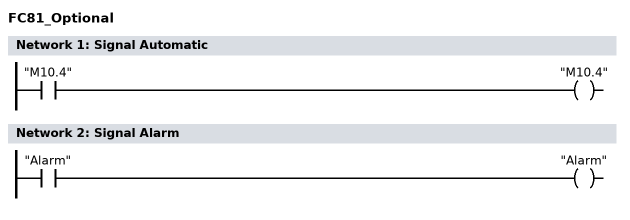
   RUNG wire#powerrail
      Contact( "M10.4" )
      Coil( "M10.4" )
   END_RUNG
   // the same network as SCL:
   "M10.4" := "M10.4";
END_REGION

REGION Network 2: Signal Alarm
   RUNG wire#powerrail
      Contact( "Alarm" )
      Coil( "Alarm" )
   END_RUNG
   // the same network as SCL:
   "Alarm" := "Alarm";
END_REGION
END_FUNCTION

FUNCTION "FC82_Conveyor_2_IN_2_OUT" : Void   // FC82, LAD
TITLE = Conveyor_2_IN_2_OUT
{ S7_Optimized_Access := 'TRUE' }
VERSION : 0.1
// stored: AutoNumber false, IsIECCheckEnabled false, SetENOAutomatically false, UDAEnableTagReadback false
   VAR_TEMP   // added for the SCL form of the ladder/FBD networks
      _w1 : Bool;
      _w2 : Bool;
   END_VAR
BEGIN

REGION Network 1: Manual operation for conveyor
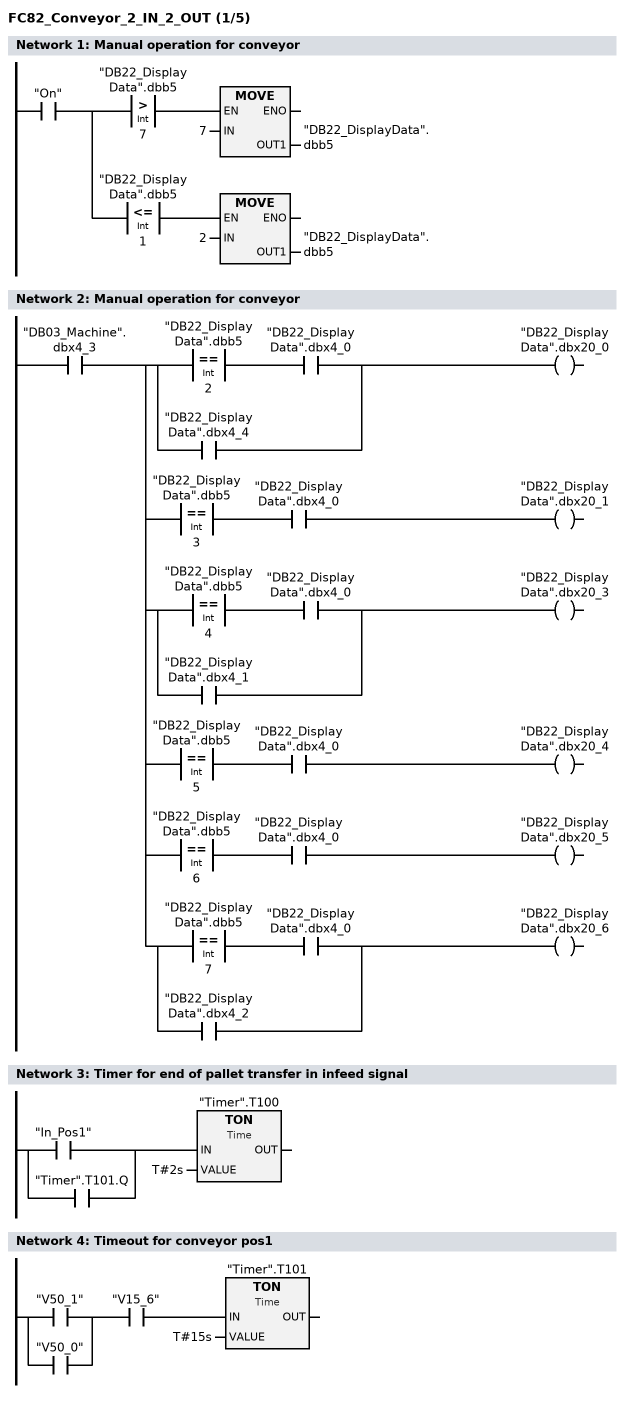
   RUNG wire#powerrail
      Contact( "On" )
      wire#w1
      { S7_Templates := "SrcType := Int" } GT_Contact(in1 := "DB22_DisplayData".dbb5, in2 := 7)
      { S7_GenerateENO := "TRUE" } Move(in := 7, out1 => "DB22_DisplayData".dbb5)
   END_RUNG
   RUNG wire#w1
      { S7_Templates := "SrcType := Int" } LE_Contact(in1 := "DB22_DisplayData".dbb5, in2 := 1)
      { S7_GenerateENO := "TRUE" } Move(in := 2, out1 => "DB22_DisplayData".dbb5)
   END_RUNG
   // the same network as SCL:
   IF "On" AND ("DB22_DisplayData".dbb5 > 7) THEN "DB22_DisplayData".dbb5 := 7; END_IF;
   IF "On" AND ("DB22_DisplayData".dbb5 <= 1) THEN "DB22_DisplayData".dbb5 := 2; END_IF;
END_REGION

REGION Network 2: Manual operation for conveyor
   RUNG wire#powerrail
      Contact( "DB03_Machine".dbx4_3 )
      wire#w1
      { S7_Templates := "SrcType := Int" } EQ_Contact(in1 := "DB22_DisplayData".dbb5, in2 := 2)
      Contact( "DB22_DisplayData".dbx4_0 )
      wire#w2
      Coil( "DB22_DisplayData".dbx20_0 )
   END_RUNG
   RUNG wire#w1
      Contact( "DB22_DisplayData".dbx4_4 )
   END_RUNG wire#w2
   RUNG wire#w1
      { S7_Templates := "SrcType := Int" } EQ_Contact(in1 := "DB22_DisplayData".dbb5, in2 := 3)
      Contact( "DB22_DisplayData".dbx4_0 )
      Coil( "DB22_DisplayData".dbx20_1 )
   END_RUNG
   RUNG wire#w1
      { S7_Templates := "SrcType := Int" } EQ_Contact(in1 := "DB22_DisplayData".dbb5, in2 := 4)
      Contact( "DB22_DisplayData".dbx4_0 )
      wire#w3
      Coil( "DB22_DisplayData".dbx20_3 )
   END_RUNG
   RUNG wire#w1
      Contact( "DB22_DisplayData".dbx4_1 )
   END_RUNG wire#w3
   RUNG wire#w1
      { S7_Templates := "SrcType := Int" } EQ_Contact(in1 := "DB22_DisplayData".dbb5, in2 := 5)
      Contact( "DB22_DisplayData".dbx4_0 )
      Coil( "DB22_DisplayData".dbx20_4 )
   END_RUNG
   RUNG wire#w1
      { S7_Templates := "SrcType := Int" } EQ_Contact(in1 := "DB22_DisplayData".dbb5, in2 := 6)
      Contact( "DB22_DisplayData".dbx4_0 )
      Coil( "DB22_DisplayData".dbx20_5 )
   END_RUNG
   RUNG wire#w1
      { S7_Templates := "SrcType := Int" } EQ_Contact(in1 := "DB22_DisplayData".dbb5, in2 := 7)
      Contact( "DB22_DisplayData".dbx4_0 )
      wire#w4
      Coil( "DB22_DisplayData".dbx20_6 )
   END_RUNG
   RUNG wire#w1
      Contact( "DB22_DisplayData".dbx4_2 )
   END_RUNG wire#w4
   // the same network as SCL:
   "DB22_DisplayData".dbx20_0 := "DB03_Machine".dbx4_3 AND ((("DB22_DisplayData".dbb5 = 2) AND "DB22_DisplayData".dbx4_0) OR "DB22_DisplayData".dbx4_4);
   "DB22_DisplayData".dbx20_1 := "DB03_Machine".dbx4_3 AND ("DB22_DisplayData".dbb5 = 3) AND "DB22_DisplayData".dbx4_0;
   "DB22_DisplayData".dbx20_3 := "DB03_Machine".dbx4_3 AND ((("DB22_DisplayData".dbb5 = 4) AND "DB22_DisplayData".dbx4_0) OR "DB22_DisplayData".dbx4_1);
   "DB22_DisplayData".dbx20_4 := "DB03_Machine".dbx4_3 AND ("DB22_DisplayData".dbb5 = 5) AND "DB22_DisplayData".dbx4_0;
   "DB22_DisplayData".dbx20_5 := "DB03_Machine".dbx4_3 AND ("DB22_DisplayData".dbb5 = 6) AND "DB22_DisplayData".dbx4_0;
   "DB22_DisplayData".dbx20_6 := "DB03_Machine".dbx4_3 AND ((("DB22_DisplayData".dbb5 = 7) AND "DB22_DisplayData".dbx4_0) OR "DB22_DisplayData".dbx4_2);
END_REGION

REGION Network 3: Timer for end of pallet transfer in infeed signal
   "Timer".T100.TON(IN := "In_Pos1" OR "Timer".T101.Q, PT := T#2s);   // TON coil
END_REGION

REGION Network 4: Timeout for conveyor pos1
   "Timer".T101.TON(IN := ("V50_1" OR "V50_0") AND "V15_6", PT := T#15s);   // TON coil
END_REGION

REGION Network 5: Time to load with forklift
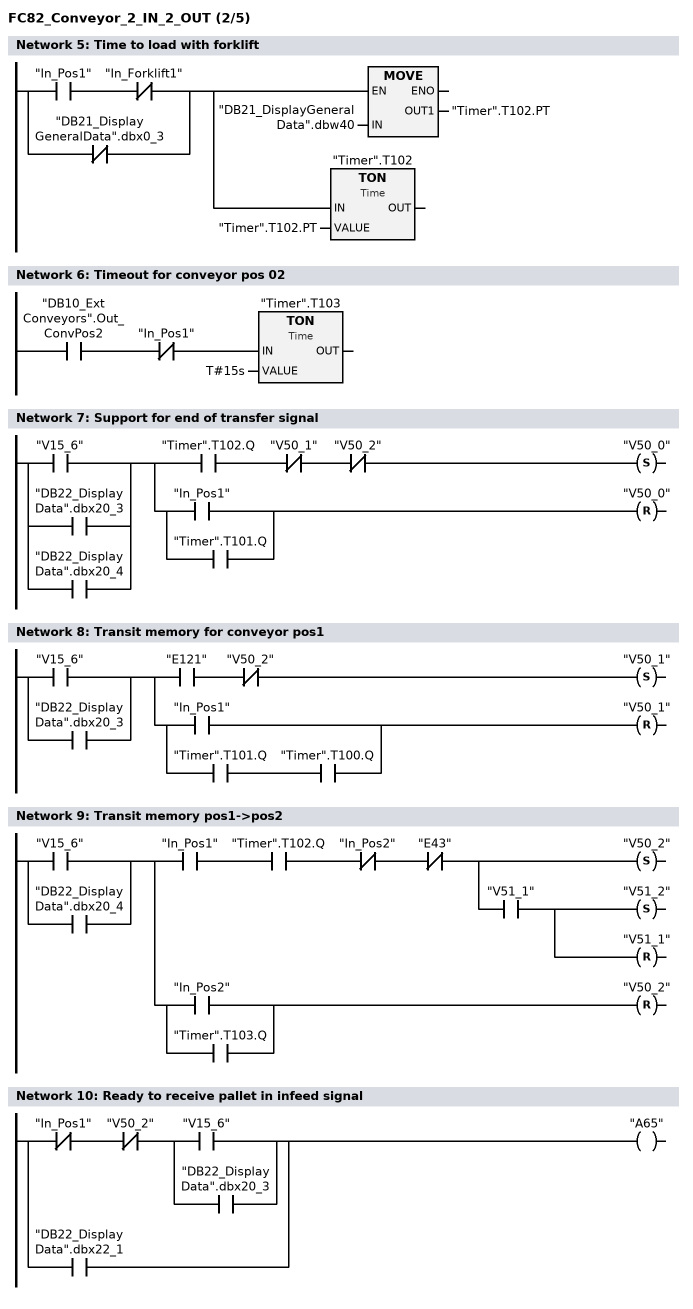
   #_w1 := ("In_Pos1" AND NOT "In_Forklift1") OR NOT "DB21_DisplayGeneralData".dbx0_3;
   IF #_w1 THEN "Timer".T102.PT := "DB21_DisplayGeneralData".dbw40; END_IF;
   "Timer".T102.TON(IN := #_w1, PT := "Timer".T102.PT);   // TON coil
END_REGION

REGION Network 6: Timeout for conveyor pos 02
   "Timer".T103.TON(IN := "DB10_ExtConveyors".Out_ConvPos2 AND NOT "In_Pos1", PT := T#15s);   // TON coil
END_REGION

REGION Network 7: Support for end of transfer signal
   RUNG wire#powerrail
      Contact( "V15_6" )
      wire#w1
      Contact( "Timer".T102.Q )
      I_Contact( "V50_1" )
      I_Contact( "V50_2" )
      S_Coil( "V50_0" )
   END_RUNG
   RUNG wire#powerrail
      Contact( "DB22_DisplayData".dbx20_3 )
   END_RUNG wire#w1
   RUNG wire#powerrail
      Contact( "DB22_DisplayData".dbx20_4 )
   END_RUNG wire#w1
   RUNG wire#w1
      Contact( "In_Pos1" )
      wire#w2
      R_Coil( "V50_0" )
   END_RUNG
   RUNG wire#w1
      Contact( "Timer".T101.Q )
   END_RUNG wire#w2
   // the same network as SCL:
   #_w1 := "V15_6" OR "DB22_DisplayData".dbx20_3 OR "DB22_DisplayData".dbx20_4;
   IF #_w1 AND "Timer".T102.Q AND NOT "V50_1" AND NOT "V50_2" THEN "V50_0" := TRUE; END_IF;
   IF #_w1 AND ("In_Pos1" OR "Timer".T101.Q) THEN "V50_0" := FALSE; END_IF;
END_REGION

REGION Network 8: Transit memory for conveyor pos1
   RUNG wire#powerrail
      Contact( "V15_6" )
      wire#w1
      Contact( "E121" )
      I_Contact( "V50_2" )
      S_Coil( "V50_1" )
   END_RUNG
   RUNG wire#powerrail
      Contact( "DB22_DisplayData".dbx20_3 )
   END_RUNG wire#w1
   RUNG wire#w1
      Contact( "In_Pos1" )
      wire#w2
      R_Coil( "V50_1" )
   END_RUNG
   RUNG wire#w1
      Contact( "Timer".T101.Q )
      Contact( "Timer".T100.Q )
   END_RUNG wire#w2
   // the same network as SCL:
   #_w1 := "V15_6" OR "DB22_DisplayData".dbx20_3;
   IF #_w1 AND "E121" AND NOT "V50_2" THEN "V50_1" := TRUE; END_IF;
   IF #_w1 AND ("In_Pos1" OR ("Timer".T101.Q AND "Timer".T100.Q)) THEN "V50_1" := FALSE; END_IF;
END_REGION

REGION Network 9: Transit memory pos1->pos2
   RUNG wire#powerrail
      Contact( "V15_6" )
      wire#w1
      Contact( "In_Pos1" )
      Contact( "Timer".T102.Q )
      I_Contact( "In_Pos2" )
      I_Contact( "E43" )
      wire#w2
      S_Coil( "V50_2" )
   END_RUNG
   RUNG wire#powerrail
      Contact( "DB22_DisplayData".dbx20_4 )
   END_RUNG wire#w1
   RUNG wire#w2
      Contact( "V51_1" )
      wire#w3
      S_Coil( "V51_2" )
   END_RUNG
   RUNG wire#w3
      R_Coil( "V51_1" )
   END_RUNG
   RUNG wire#w1
      Contact( "In_Pos2" )
      wire#w4
      R_Coil( "V50_2" )
   END_RUNG
   RUNG wire#w1
      Contact( "Timer".T103.Q )
   END_RUNG wire#w4
   // the same network as SCL:
   #_w1 := "V15_6" OR "DB22_DisplayData".dbx20_4;
   #_w2 := #_w1 AND "In_Pos1" AND "Timer".T102.Q AND NOT "In_Pos2" AND NOT "E43";
   IF #_w2 THEN "V50_2" := TRUE; END_IF;
   IF #_w2 AND "V51_1" THEN
       "V51_2" := TRUE;
       "V51_1" := FALSE;
   END_IF;
   IF #_w1 AND ("In_Pos2" OR "Timer".T103.Q) THEN "V50_2" := FALSE; END_IF;
END_REGION

REGION Network 10: Ready to receive pallet in infeed signal
   RUNG wire#powerrail
      I_Contact( "In_Pos1" )
      I_Contact( "V50_2" )
      wire#w1
      Contact( "V15_6" )
      wire#w2
      Coil( "A65" )
   END_RUNG
   RUNG wire#w1
      Contact( "DB22_DisplayData".dbx20_3 )
   END_RUNG wire#w2
   RUNG wire#powerrail
      Contact( "DB22_DisplayData".dbx22_1 )
   END_RUNG wire#w2
   // the same network as SCL:
   "A65" := (NOT "In_Pos1" AND NOT "V50_2" AND ("V15_6" OR "DB22_DisplayData".dbx20_3)) OR "DB22_DisplayData".dbx22_1;
END_REGION

REGION Network 11: End of pallet transfer in infeed signal
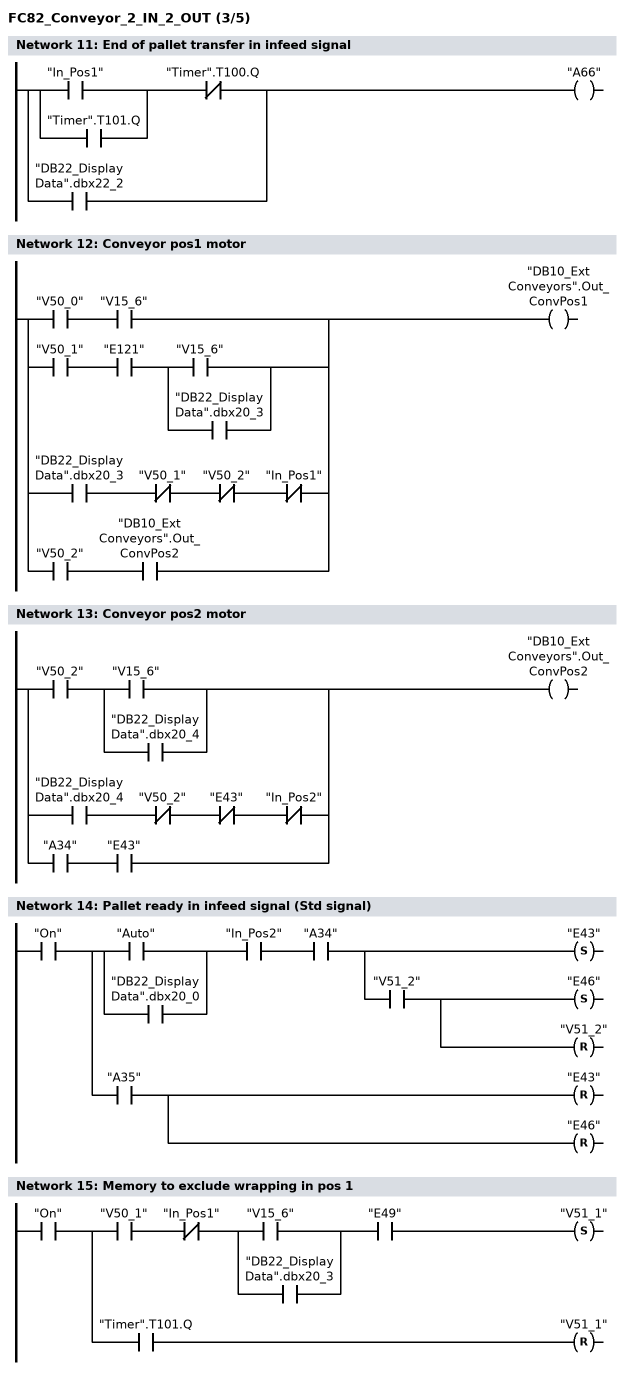
   RUNG wire#powerrail
      Contact( "In_Pos1" )
      wire#w1
      I_Contact( "Timer".T100.Q )
      wire#w2
      Coil( "A66" )
   END_RUNG
   RUNG wire#powerrail
      Contact( "Timer".T101.Q )
   END_RUNG wire#w1
   RUNG wire#powerrail
      Contact( "DB22_DisplayData".dbx22_2 )
   END_RUNG wire#w2
   // the same network as SCL:
   "A66" := (("In_Pos1" OR "Timer".T101.Q) AND NOT "Timer".T100.Q) OR "DB22_DisplayData".dbx22_2;
END_REGION

REGION Network 12: Conveyor pos1 motor
   RUNG wire#powerrail
      Contact( "V50_0" )
      Contact( "V15_6" )
      wire#w1
      Coil( "DB10_ExtConveyors".Out_ConvPos1 )
   END_RUNG
   RUNG wire#powerrail
      Contact( "V50_1" )
      Contact( "E121" )
      wire#w2
      Contact( "V15_6" )
   END_RUNG wire#w1
   RUNG wire#w2
      Contact( "DB22_DisplayData".dbx20_3 )
   END_RUNG wire#w1
   RUNG wire#powerrail
      Contact( "DB22_DisplayData".dbx20_3 )
      I_Contact( "V50_1" )
      I_Contact( "V50_2" )
      I_Contact( "In_Pos1" )
   END_RUNG wire#w1
   RUNG wire#powerrail
      Contact( "V50_2" )
      Contact( "DB10_ExtConveyors".Out_ConvPos2 )
   END_RUNG wire#w1
   // the same network as SCL:
   "DB10_ExtConveyors".Out_ConvPos1 := ("V50_0" AND "V15_6") OR ("V50_1" AND "E121" AND ("V15_6" OR "DB22_DisplayData".dbx20_3)) OR ("DB22_DisplayData".dbx20_3 AND NOT "V50_1" AND NOT "V50_2" AND NOT "In_Pos1") OR ("V50_2" AND "DB10_ExtConveyors".Out_ConvPos2);
END_REGION

REGION Network 13: Conveyor pos2 motor
   RUNG wire#powerrail
      Contact( "V50_2" )
      wire#w1
      Contact( "V15_6" )
      wire#w2
      Coil( "DB10_ExtConveyors".Out_ConvPos2 )
   END_RUNG
   RUNG wire#w1
      Contact( "DB22_DisplayData".dbx20_4 )
   END_RUNG wire#w2
   RUNG wire#powerrail
      Contact( "DB22_DisplayData".dbx20_4 )
      I_Contact( "V50_2" )
      I_Contact( "E43" )
      I_Contact( "In_Pos2" )
   END_RUNG wire#w2
   RUNG wire#powerrail
      Contact( "A34" )
      Contact( "E43" )
   END_RUNG wire#w2
   // the same network as SCL:
   "DB10_ExtConveyors".Out_ConvPos2 := ("V50_2" AND ("V15_6" OR "DB22_DisplayData".dbx20_4)) OR ("DB22_DisplayData".dbx20_4 AND NOT "V50_2" AND NOT "E43" AND NOT "In_Pos2") OR ("A34" AND "E43");
END_REGION

REGION Network 14: Pallet ready in infeed signal (Std signal)
   RUNG wire#powerrail
      Contact( "On" )
      wire#w1
      Contact( "Auto" )
      wire#w2
      Contact( "In_Pos2" )
      Contact( "A34" )
      wire#w3
      S_Coil( "E43" )
   END_RUNG
   RUNG wire#w1
      Contact( "DB22_DisplayData".dbx20_0 )
   END_RUNG wire#w2
   RUNG wire#w3
      Contact( "V51_2" )
      wire#w4
      S_Coil( "E46" )
   END_RUNG
   RUNG wire#w4
      R_Coil( "V51_2" )
   END_RUNG
   RUNG wire#w1
      Contact( "A35" )
      wire#w5
      R_Coil( "E43" )
   END_RUNG
   RUNG wire#w5
      R_Coil( "E46" )
   END_RUNG
   // the same network as SCL:
   #_w1 := "On" AND ("Auto" OR "DB22_DisplayData".dbx20_0) AND "In_Pos2" AND "A34";
   IF #_w1 THEN "E43" := TRUE; END_IF;
   IF #_w1 AND "V51_2" THEN
       "E46" := TRUE;
       "V51_2" := FALSE;
   END_IF;
   IF "On" AND "A35" THEN
       "E43" := FALSE;
       "E46" := FALSE;
   END_IF;
END_REGION

REGION Network 15: Memory to exclude wrapping in pos 1
   RUNG wire#powerrail
      Contact( "On" )
      wire#w1
      Contact( "V50_1" )
      I_Contact( "In_Pos1" )
      wire#w2
      Contact( "V15_6" )
      wire#w3
      Contact( "E49" )
      S_Coil( "V51_1" )
   END_RUNG
   RUNG wire#w2
      Contact( "DB22_DisplayData".dbx20_3 )
   END_RUNG wire#w3
   RUNG wire#w1
      Contact( "Timer".T101.Q )
      R_Coil( "V51_1" )
   END_RUNG
   // the same network as SCL:
   IF "On" AND "V50_1" AND NOT "In_Pos1" AND ("V15_6" OR "DB22_DisplayData".dbx20_3) AND "E49" THEN
       "V51_1" := TRUE;
   END_IF;
   IF "On" AND "Timer".T101.Q THEN "V51_1" := FALSE; END_IF;
END_REGION

REGION Network 16: Conveyor pos1 motor speed selection
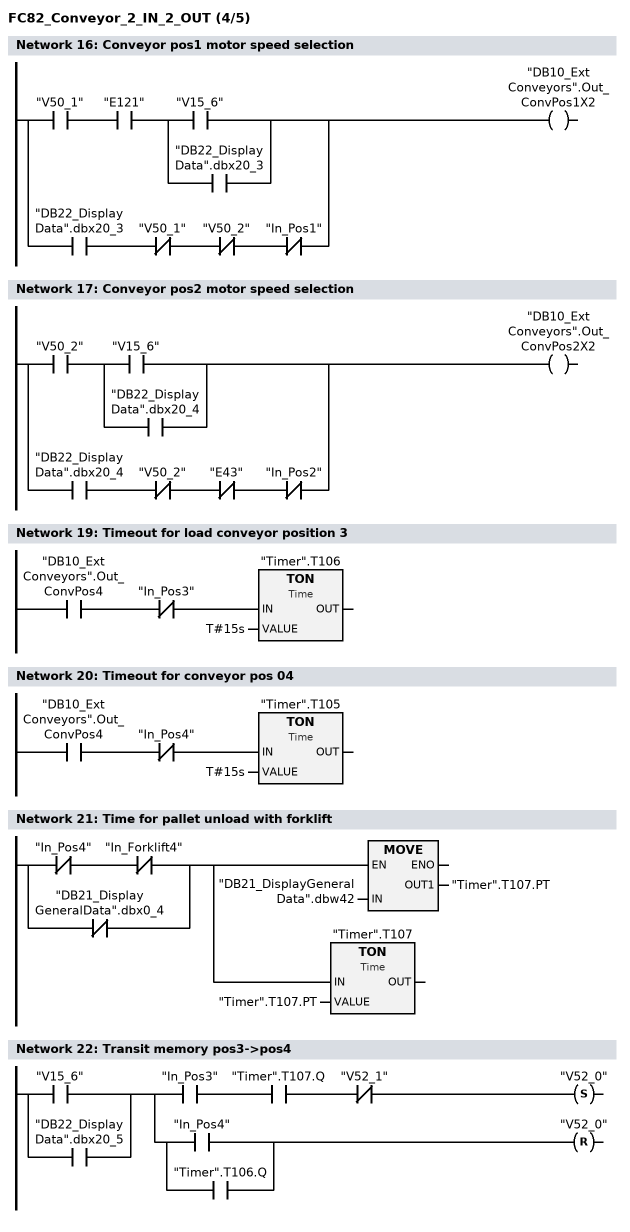
   RUNG wire#powerrail
      Contact( "V50_1" )
      Contact( "E121" )
      wire#w1
      Contact( "V15_6" )
      wire#w2
      Coil( "DB10_ExtConveyors".Out_ConvPos1X2 )
   END_RUNG
   RUNG wire#w1
      Contact( "DB22_DisplayData".dbx20_3 )
   END_RUNG wire#w2
   RUNG wire#powerrail
      Contact( "DB22_DisplayData".dbx20_3 )
      I_Contact( "V50_1" )
      I_Contact( "V50_2" )
      I_Contact( "In_Pos1" )
   END_RUNG wire#w2
   // the same network as SCL:
   "DB10_ExtConveyors".Out_ConvPos1X2 := ("V50_1" AND "E121" AND ("V15_6" OR "DB22_DisplayData".dbx20_3)) OR ("DB22_DisplayData".dbx20_3 AND NOT "V50_1" AND NOT "V50_2" AND NOT "In_Pos1");
END_REGION

REGION Network 17: Conveyor pos2 motor speed selection
   RUNG wire#powerrail
      Contact( "V50_2" )
      wire#w1
      Contact( "V15_6" )
      wire#w2
      Coil( "DB10_ExtConveyors".Out_ConvPos2X2 )
   END_RUNG
   RUNG wire#w1
      Contact( "DB22_DisplayData".dbx20_4 )
   END_RUNG wire#w2
   RUNG wire#powerrail
      Contact( "DB22_DisplayData".dbx20_4 )
      I_Contact( "V50_2" )
      I_Contact( "E43" )
      I_Contact( "In_Pos2" )
   END_RUNG wire#w2
   // the same network as SCL:
   "DB10_ExtConveyors".Out_ConvPos2X2 := ("V50_2" AND ("V15_6" OR "DB22_DisplayData".dbx20_4)) OR ("DB22_DisplayData".dbx20_4 AND NOT "V50_2" AND NOT "E43" AND NOT "In_Pos2");
END_REGION

REGION Network 18: >>>>>>> OUTFEED CONVEYORS <<<<<<<<
END_REGION

REGION Network 19: Timeout for load conveyor position 3
   "Timer".T106.TON(IN := "DB10_ExtConveyors".Out_ConvPos4 AND NOT "In_Pos3", PT := T#15s);   // TON coil
END_REGION

REGION Network 20: Timeout for conveyor pos 04
   "Timer".T105.TON(IN := "DB10_ExtConveyors".Out_ConvPos4 AND NOT "In_Pos4", PT := T#15s);   // TON coil
END_REGION

REGION Network 21: Time for pallet unload with forklift
   #_w1 := (NOT "In_Pos4" AND NOT "In_Forklift4") OR NOT "DB21_DisplayGeneralData".dbx0_4;
   IF #_w1 THEN "Timer".T107.PT := "DB21_DisplayGeneralData".dbw42; END_IF;
   "Timer".T107.TON(IN := #_w1, PT := "Timer".T107.PT);   // TON coil
END_REGION

REGION Network 22: Transit memory pos3->pos4
   RUNG wire#powerrail
      Contact( "V15_6" )
      wire#w1
      Contact( "In_Pos3" )
      Contact( "Timer".T107.Q )
      I_Contact( "V52_1" )
      S_Coil( "V52_0" )
   END_RUNG
   RUNG wire#powerrail
      Contact( "DB22_DisplayData".dbx20_5 )
   END_RUNG wire#w1
   RUNG wire#w1
      Contact( "In_Pos4" )
      wire#w2
      R_Coil( "V52_0" )
   END_RUNG
   RUNG wire#w1
      Contact( "Timer".T106.Q )
   END_RUNG wire#w2
   // the same network as SCL:
   #_w1 := "V15_6" OR "DB22_DisplayData".dbx20_5;
   IF #_w1 AND "In_Pos3" AND "Timer".T107.Q AND NOT "V52_1" THEN "V52_0" := TRUE; END_IF;
   IF #_w1 AND ("In_Pos4" OR "Timer".T106.Q) THEN "V52_0" := FALSE; END_IF;
END_REGION

REGION Network 23: Outfeed conveyor pos.4 unload
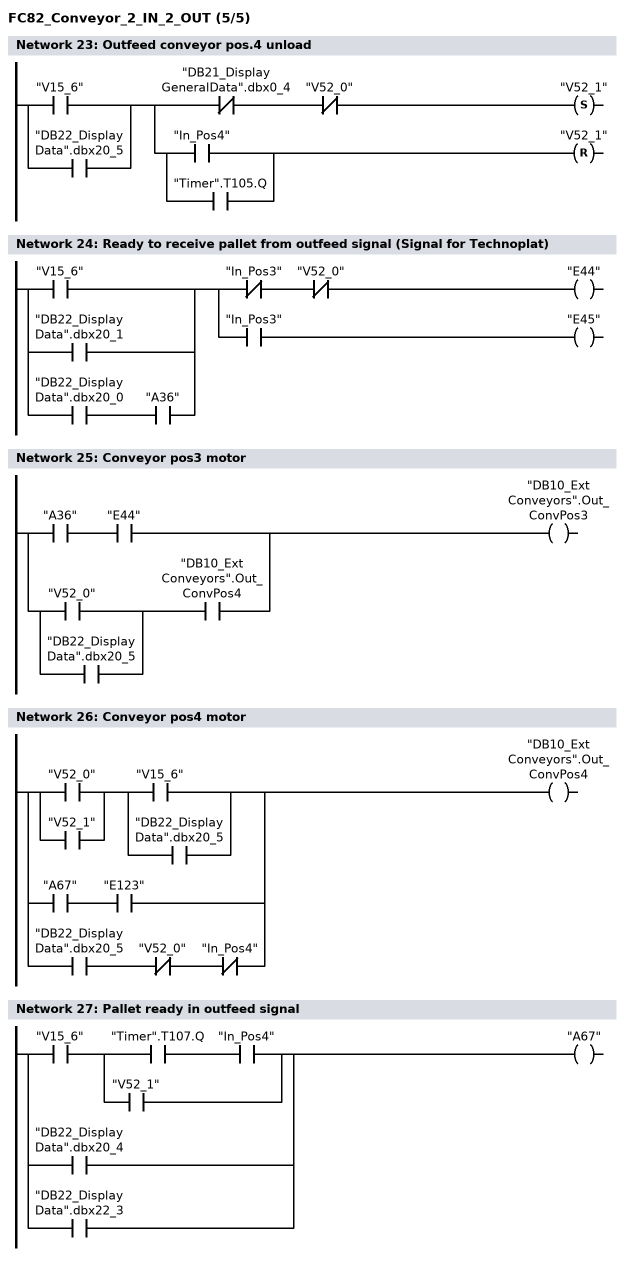
   RUNG wire#powerrail
      Contact( "V15_6" )
      wire#w1
      I_Contact( "DB21_DisplayGeneralData".dbx0_4 )
      I_Contact( "V52_0" )
      S_Coil( "V52_1" )
   END_RUNG
   RUNG wire#powerrail
      Contact( "DB22_DisplayData".dbx20_5 )
   END_RUNG wire#w1
   RUNG wire#w1
      Contact( "In_Pos4" )
      wire#w2
      R_Coil( "V52_1" )
   END_RUNG
   RUNG wire#w1
      Contact( "Timer".T105.Q )
   END_RUNG wire#w2
   // the same network as SCL:
   #_w1 := "V15_6" OR "DB22_DisplayData".dbx20_5;
   IF #_w1 AND NOT "DB21_DisplayGeneralData".dbx0_4 AND NOT "V52_0" THEN "V52_1" := TRUE; END_IF;
   IF #_w1 AND ("In_Pos4" OR "Timer".T105.Q) THEN "V52_1" := FALSE; END_IF;
END_REGION

REGION Network 24: Ready to receive pallet from outfeed signal (Signal for Technoplat)
   RUNG wire#powerrail
      Contact( "V15_6" )
      wire#w1
      I_Contact( "In_Pos3" )
      I_Contact( "V52_0" )
      Coil( "E44" )
   END_RUNG
   RUNG wire#powerrail
      Contact( "DB22_DisplayData".dbx20_1 )
   END_RUNG wire#w1
   RUNG wire#powerrail
      Contact( "DB22_DisplayData".dbx20_0 )
      Contact( "A36" )
   END_RUNG wire#w1
   RUNG wire#w1
      Contact( "In_Pos3" )
      Coil( "E45" )
   END_RUNG
   // the same network as SCL:
   #_w1 := "V15_6" OR "DB22_DisplayData".dbx20_1 OR ("DB22_DisplayData".dbx20_0 AND "A36");
   "E44" := #_w1 AND NOT "In_Pos3" AND NOT "V52_0";
   "E45" := #_w1 AND "In_Pos3";
END_REGION

REGION Network 25: Conveyor pos3 motor
   RUNG wire#powerrail
      Contact( "A36" )
      Contact( "E44" )
      wire#w1
      Coil( "DB10_ExtConveyors".Out_ConvPos3 )
   END_RUNG
   RUNG wire#powerrail
      Contact( "V52_0" )
      wire#w2
      Contact( "DB10_ExtConveyors".Out_ConvPos4 )
   END_RUNG wire#w1
   RUNG wire#powerrail
      Contact( "DB22_DisplayData".dbx20_5 )
   END_RUNG wire#w2
   // the same network as SCL:
   "DB10_ExtConveyors".Out_ConvPos3 := ("A36" AND "E44") OR (("V52_0" OR "DB22_DisplayData".dbx20_5) AND "DB10_ExtConveyors".Out_ConvPos4);
END_REGION

REGION Network 26: Conveyor pos4 motor
   RUNG wire#powerrail
      Contact( "V52_0" )
      wire#w1
      Contact( "V15_6" )
      wire#w2
      Coil( "DB10_ExtConveyors".Out_ConvPos4 )
   END_RUNG
   RUNG wire#powerrail
      Contact( "V52_1" )
   END_RUNG wire#w1
   RUNG wire#w1
      Contact( "DB22_DisplayData".dbx20_5 )
   END_RUNG wire#w2
   RUNG wire#powerrail
      Contact( "A67" )
      Contact( "E123" )
   END_RUNG wire#w2
   RUNG wire#powerrail
      Contact( "DB22_DisplayData".dbx20_5 )
      I_Contact( "V52_0" )
      I_Contact( "In_Pos4" )
   END_RUNG wire#w2
   // the same network as SCL:
   "DB10_ExtConveyors".Out_ConvPos4 := (("V52_0" OR "V52_1") AND ("V15_6" OR "DB22_DisplayData".dbx20_5)) OR ("A67" AND "E123") OR ("DB22_DisplayData".dbx20_5 AND NOT "V52_0" AND NOT "In_Pos4");
END_REGION

REGION Network 27: Pallet ready in outfeed signal
   RUNG wire#powerrail
      Contact( "V15_6" )
      wire#w1
      Contact( "Timer".T107.Q )
      Contact( "In_Pos4" )
      wire#w2
      Coil( "A67" )
   END_RUNG
   RUNG wire#w1
      Contact( "V52_1" )
   END_RUNG wire#w2
   RUNG wire#powerrail
      Contact( "DB22_DisplayData".dbx20_4 )
   END_RUNG wire#w2
   RUNG wire#powerrail
      Contact( "DB22_DisplayData".dbx22_3 )
   END_RUNG wire#w2
   // the same network as SCL:
   "A67" := ("V15_6" AND (("Timer".T107.Q AND "In_Pos4") OR "V52_1")) OR "DB22_DisplayData".dbx20_4 OR "DB22_DisplayData".dbx22_3;
END_REGION
END_FUNCTION

FUNCTION "FC90_PageManagement" : Void   // FC90, LAD
{ S7_Optimized_Access := 'FALSE' }
VERSION : 0.1
// stored: AutoNumber false, IsIECCheckEnabled false, SetENOAutomatically false, UDAEnableTagReadback false
   VAR_TEMP
      CurrentPage : Int;
      PageBkwRequest : Int;
      PageFwRequest : Int;
   END_VAR
   VAR_TEMP   // added for the SCL form of the ladder/FBD networks
      _w1 : Bool;
   END_VAR
BEGIN

REGION Network 1
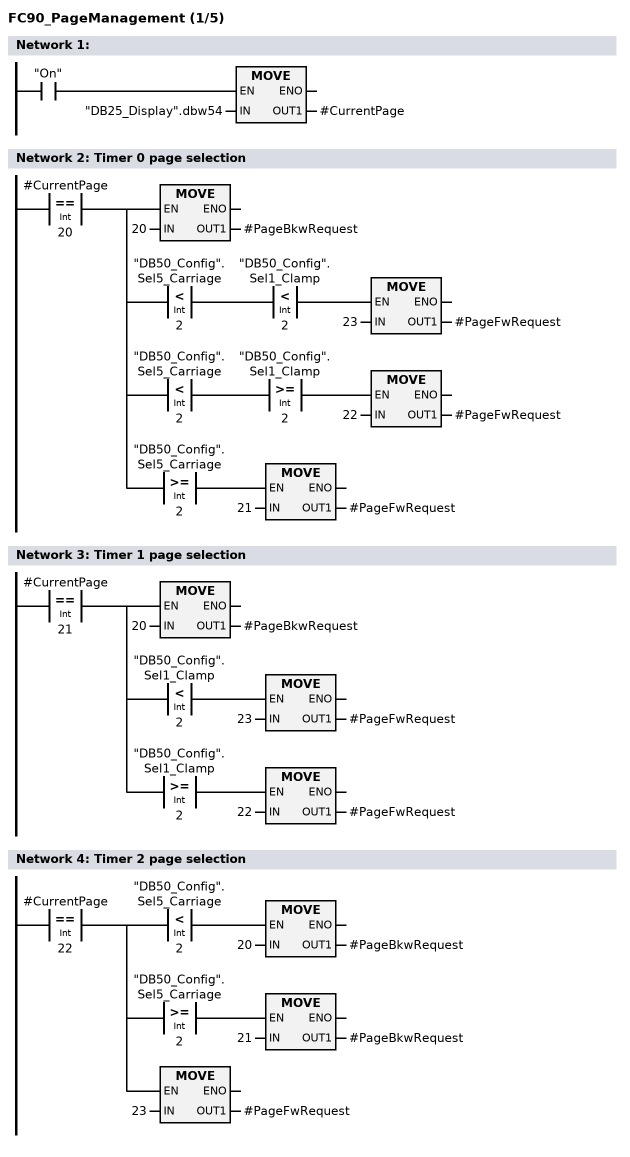
   RUNG wire#powerrail
      Contact( "On" )
      { S7_GenerateENO := "TRUE" } Move(in := "DB25_Display".dbw54, out1 => #CurrentPage)
   END_RUNG
   // the same network as SCL:
   IF "On" THEN #CurrentPage := "DB25_Display".dbw54; END_IF;
END_REGION

REGION Network 2: Timer 0 page selection
   RUNG wire#powerrail
      { S7_Templates := "SrcType := Int" } EQ_Contact(in1 := #CurrentPage, in2 := 20)
      wire#w1
      { S7_GenerateENO := "TRUE" } Move(in := 20, out1 => #PageBkwRequest)
   END_RUNG
   RUNG wire#w1
      { S7_Templates := "SrcType := Int" } LT_Contact(in1 := "DB50_Config".Sel5_Carriage, in2 := 2)
      { S7_Templates := "SrcType := Int" } LT_Contact(in1 := "DB50_Config".Sel1_Clamp, in2 := 2)
      { S7_GenerateENO := "TRUE" } Move(in := 23, out1 => #PageFwRequest)
   END_RUNG
   RUNG wire#w1
      { S7_Templates := "SrcType := Int" } LT_Contact(in1 := "DB50_Config".Sel5_Carriage, in2 := 2)
      { S7_Templates := "SrcType := Int" } GE_Contact(in1 := "DB50_Config".Sel1_Clamp, in2 := 2)
      { S7_GenerateENO := "TRUE" } Move(in := 22, out1 => #PageFwRequest)
   END_RUNG
   RUNG wire#w1
      { S7_Templates := "SrcType := Int" } GE_Contact(in1 := "DB50_Config".Sel5_Carriage, in2 := 2)
      { S7_GenerateENO := "TRUE" } Move(in := 21, out1 => #PageFwRequest)
   END_RUNG
   // the same network as SCL:
   #_w1 := #CurrentPage = 20;
   IF #_w1 THEN #PageBkwRequest := 20; END_IF;
   IF #_w1 AND ("DB50_Config".Sel5_Carriage < 2) AND ("DB50_Config".Sel1_Clamp < 2) THEN
       #PageFwRequest := 23;
   END_IF;
   IF #_w1 AND ("DB50_Config".Sel5_Carriage < 2) AND ("DB50_Config".Sel1_Clamp >= 2) THEN
       #PageFwRequest := 22;
   END_IF;
   IF #_w1 AND ("DB50_Config".Sel5_Carriage >= 2) THEN #PageFwRequest := 21; END_IF;
END_REGION

REGION Network 3: Timer 1 page selection
   RUNG wire#powerrail
      { S7_Templates := "SrcType := Int" } EQ_Contact(in1 := #CurrentPage, in2 := 21)
      wire#w1
      { S7_GenerateENO := "TRUE" } Move(in := 20, out1 => #PageBkwRequest)
   END_RUNG
   RUNG wire#w1
      { S7_Templates := "SrcType := Int" } LT_Contact(in1 := "DB50_Config".Sel1_Clamp, in2 := 2)
      { S7_GenerateENO := "TRUE" } Move(in := 23, out1 => #PageFwRequest)
   END_RUNG
   RUNG wire#w1
      { S7_Templates := "SrcType := Int" } GE_Contact(in1 := "DB50_Config".Sel1_Clamp, in2 := 2)
      { S7_GenerateENO := "TRUE" } Move(in := 22, out1 => #PageFwRequest)
   END_RUNG
   // the same network as SCL:
   #_w1 := #CurrentPage = 21;
   IF #_w1 THEN #PageBkwRequest := 20; END_IF;
   IF #_w1 AND ("DB50_Config".Sel1_Clamp < 2) THEN #PageFwRequest := 23; END_IF;
   IF #_w1 AND ("DB50_Config".Sel1_Clamp >= 2) THEN #PageFwRequest := 22; END_IF;
END_REGION

REGION Network 4: Timer 2 page selection
   RUNG wire#powerrail
      { S7_Templates := "SrcType := Int" } EQ_Contact(in1 := #CurrentPage, in2 := 22)
      wire#w1
      { S7_Templates := "SrcType := Int" } LT_Contact(in1 := "DB50_Config".Sel5_Carriage, in2 := 2)
      { S7_GenerateENO := "TRUE" } Move(in := 20, out1 => #PageBkwRequest)
   END_RUNG
   RUNG wire#w1
      { S7_Templates := "SrcType := Int" } GE_Contact(in1 := "DB50_Config".Sel5_Carriage, in2 := 2)
      { S7_GenerateENO := "TRUE" } Move(in := 21, out1 => #PageBkwRequest)
   END_RUNG
   RUNG wire#w1
      { S7_GenerateENO := "TRUE" } Move(in := 23, out1 => #PageFwRequest)
   END_RUNG
   // the same network as SCL:
   #_w1 := #CurrentPage = 22;
   IF #_w1 AND ("DB50_Config".Sel5_Carriage < 2) THEN #PageBkwRequest := 20; END_IF;
   IF #_w1 AND ("DB50_Config".Sel5_Carriage >= 2) THEN #PageBkwRequest := 21; END_IF;
   IF #_w1 THEN #PageFwRequest := 23; END_IF;
END_REGION

REGION Network 5: Timer 3 page selection
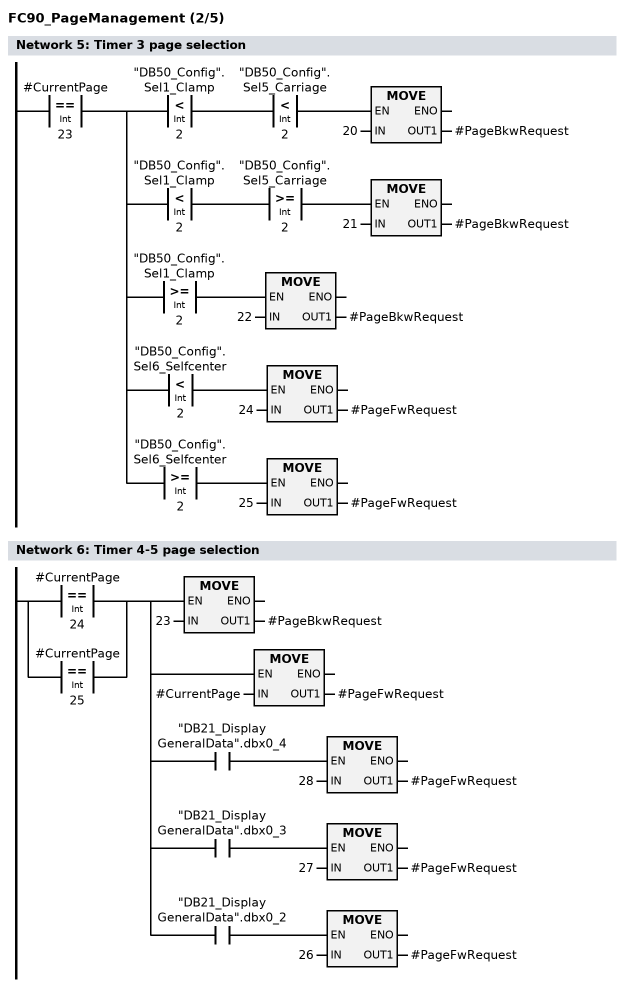
   RUNG wire#powerrail
      { S7_Templates := "SrcType := Int" } EQ_Contact(in1 := #CurrentPage, in2 := 23)
      wire#w1
      { S7_Templates := "SrcType := Int" } LT_Contact(in1 := "DB50_Config".Sel1_Clamp, in2 := 2)
      { S7_Templates := "SrcType := Int" } LT_Contact(in1 := "DB50_Config".Sel5_Carriage, in2 := 2)
      { S7_GenerateENO := "TRUE" } Move(in := 20, out1 => #PageBkwRequest)
   END_RUNG
   RUNG wire#w1
      { S7_Templates := "SrcType := Int" } LT_Contact(in1 := "DB50_Config".Sel1_Clamp, in2 := 2)
      { S7_Templates := "SrcType := Int" } GE_Contact(in1 := "DB50_Config".Sel5_Carriage, in2 := 2)
      { S7_GenerateENO := "TRUE" } Move(in := 21, out1 => #PageBkwRequest)
   END_RUNG
   RUNG wire#w1
      { S7_Templates := "SrcType := Int" } GE_Contact(in1 := "DB50_Config".Sel1_Clamp, in2 := 2)
      { S7_GenerateENO := "TRUE" } Move(in := 22, out1 => #PageBkwRequest)
   END_RUNG
   RUNG wire#w1
      { S7_Templates := "SrcType := Int" } LT_Contact(in1 := "DB50_Config".Sel6_Selfcenter, in2 := 2)
      { S7_GenerateENO := "TRUE" } Move(in := 24, out1 => #PageFwRequest)
   END_RUNG
   RUNG wire#w1
      { S7_Templates := "SrcType := Int" } GE_Contact(in1 := "DB50_Config".Sel6_Selfcenter, in2 := 2)
      { S7_GenerateENO := "TRUE" } Move(in := 25, out1 => #PageFwRequest)
   END_RUNG
   // the same network as SCL:
   #_w1 := #CurrentPage = 23;
   IF #_w1 AND ("DB50_Config".Sel1_Clamp < 2) AND ("DB50_Config".Sel5_Carriage < 2) THEN
       #PageBkwRequest := 20;
   END_IF;
   IF #_w1 AND ("DB50_Config".Sel1_Clamp < 2) AND ("DB50_Config".Sel5_Carriage >= 2) THEN
       #PageBkwRequest := 21;
   END_IF;
   IF #_w1 AND ("DB50_Config".Sel1_Clamp >= 2) THEN #PageBkwRequest := 22; END_IF;
   IF #_w1 AND ("DB50_Config".Sel6_Selfcenter < 2) THEN #PageFwRequest := 24; END_IF;
   IF #_w1 AND ("DB50_Config".Sel6_Selfcenter >= 2) THEN #PageFwRequest := 25; END_IF;
END_REGION

REGION Network 6: Timer 4-5 page selection
   RUNG wire#powerrail
      { S7_Templates := "SrcType := Int" } EQ_Contact(in1 := #CurrentPage, in2 := 24)
      wire#w1
      { S7_GenerateENO := "TRUE" } Move(in := 23, out1 => #PageBkwRequest)
   END_RUNG
   RUNG wire#powerrail
      { S7_Templates := "SrcType := Int" } EQ_Contact(in1 := #CurrentPage, in2 := 25)
   END_RUNG wire#w1
   RUNG wire#w1
      { S7_GenerateENO := "TRUE" } Move(in := #CurrentPage, out1 => #PageFwRequest)
   END_RUNG
   RUNG wire#w1
      Contact( "DB21_DisplayGeneralData".dbx0_4 )
      { S7_GenerateENO := "TRUE" } Move(in := 28, out1 => #PageFwRequest)
   END_RUNG
   RUNG wire#w1
      Contact( "DB21_DisplayGeneralData".dbx0_3 )
      { S7_GenerateENO := "TRUE" } Move(in := 27, out1 => #PageFwRequest)
   END_RUNG
   RUNG wire#w1
      Contact( "DB21_DisplayGeneralData".dbx0_2 )
      { S7_GenerateENO := "TRUE" } Move(in := 26, out1 => #PageFwRequest)
   END_RUNG
   // the same network as SCL:
   #_w1 := (#CurrentPage = 24) OR (#CurrentPage = 25);
   IF #_w1 THEN
       #PageBkwRequest := 23;
       #PageFwRequest := #CurrentPage;
   END_IF;
   IF #_w1 AND "DB21_DisplayGeneralData".dbx0_4 THEN #PageFwRequest := 28; END_IF;
   IF #_w1 AND "DB21_DisplayGeneralData".dbx0_3 THEN #PageFwRequest := 27; END_IF;
   IF #_w1 AND "DB21_DisplayGeneralData".dbx0_2 THEN #PageFwRequest := 26; END_IF;
END_REGION

REGION Network 7: Timer 6 page selection
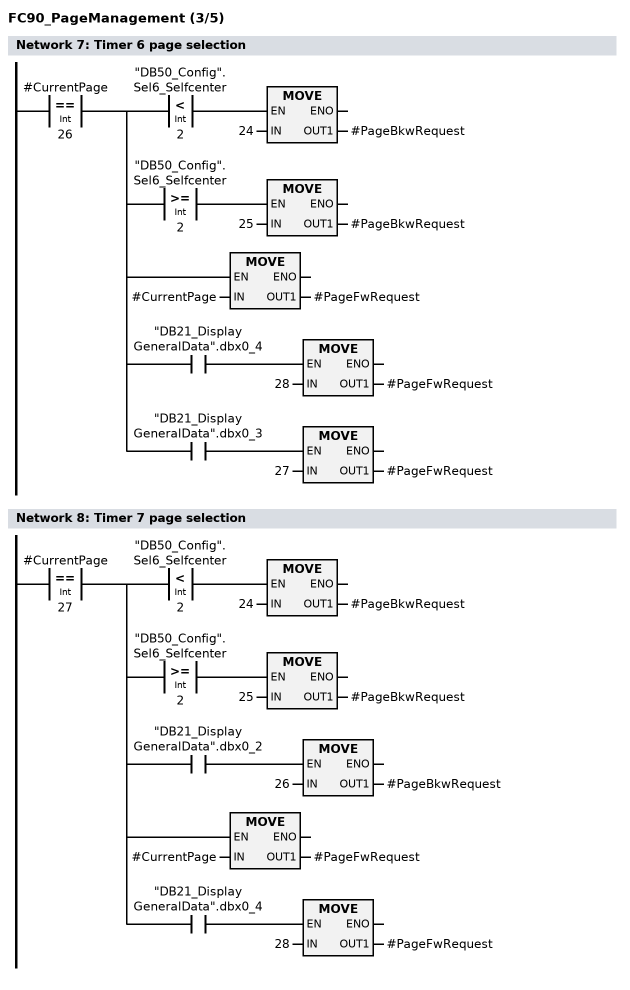
   RUNG wire#powerrail
      { S7_Templates := "SrcType := Int" } EQ_Contact(in1 := #CurrentPage, in2 := 26)
      wire#w1
      { S7_Templates := "SrcType := Int" } LT_Contact(in1 := "DB50_Config".Sel6_Selfcenter, in2 := 2)
      { S7_GenerateENO := "TRUE" } Move(in := 24, out1 => #PageBkwRequest)
   END_RUNG
   RUNG wire#w1
      { S7_Templates := "SrcType := Int" } GE_Contact(in1 := "DB50_Config".Sel6_Selfcenter, in2 := 2)
      { S7_GenerateENO := "TRUE" } Move(in := 25, out1 => #PageBkwRequest)
   END_RUNG
   RUNG wire#w1
      { S7_GenerateENO := "TRUE" } Move(in := #CurrentPage, out1 => #PageFwRequest)
   END_RUNG
   RUNG wire#w1
      Contact( "DB21_DisplayGeneralData".dbx0_4 )
      { S7_GenerateENO := "TRUE" } Move(in := 28, out1 => #PageFwRequest)
   END_RUNG
   RUNG wire#w1
      Contact( "DB21_DisplayGeneralData".dbx0_3 )
      { S7_GenerateENO := "TRUE" } Move(in := 27, out1 => #PageFwRequest)
   END_RUNG
   // the same network as SCL:
   #_w1 := #CurrentPage = 26;
   IF #_w1 AND ("DB50_Config".Sel6_Selfcenter < 2) THEN #PageBkwRequest := 24; END_IF;
   IF #_w1 AND ("DB50_Config".Sel6_Selfcenter >= 2) THEN #PageBkwRequest := 25; END_IF;
   IF #_w1 THEN #PageFwRequest := #CurrentPage; END_IF;
   IF #_w1 AND "DB21_DisplayGeneralData".dbx0_4 THEN #PageFwRequest := 28; END_IF;
   IF #_w1 AND "DB21_DisplayGeneralData".dbx0_3 THEN #PageFwRequest := 27; END_IF;
END_REGION

REGION Network 8: Timer 7 page selection
   RUNG wire#powerrail
      { S7_Templates := "SrcType := Int" } EQ_Contact(in1 := #CurrentPage, in2 := 27)
      wire#w1
      { S7_Templates := "SrcType := Int" } LT_Contact(in1 := "DB50_Config".Sel6_Selfcenter, in2 := 2)
      { S7_GenerateENO := "TRUE" } Move(in := 24, out1 => #PageBkwRequest)
   END_RUNG
   RUNG wire#w1
      { S7_Templates := "SrcType := Int" } GE_Contact(in1 := "DB50_Config".Sel6_Selfcenter, in2 := 2)
      { S7_GenerateENO := "TRUE" } Move(in := 25, out1 => #PageBkwRequest)
   END_RUNG
   RUNG wire#w1
      Contact( "DB21_DisplayGeneralData".dbx0_2 )
      { S7_GenerateENO := "TRUE" } Move(in := 26, out1 => #PageBkwRequest)
   END_RUNG
   RUNG wire#w1
      { S7_GenerateENO := "TRUE" } Move(in := #CurrentPage, out1 => #PageFwRequest)
   END_RUNG
   RUNG wire#w1
      Contact( "DB21_DisplayGeneralData".dbx0_4 )
      { S7_GenerateENO := "TRUE" } Move(in := 28, out1 => #PageFwRequest)
   END_RUNG
   // the same network as SCL:
   #_w1 := #CurrentPage = 27;
   IF #_w1 AND ("DB50_Config".Sel6_Selfcenter < 2) THEN #PageBkwRequest := 24; END_IF;
   IF #_w1 AND ("DB50_Config".Sel6_Selfcenter >= 2) THEN #PageBkwRequest := 25; END_IF;
   IF #_w1 AND "DB21_DisplayGeneralData".dbx0_2 THEN #PageBkwRequest := 26; END_IF;
   IF #_w1 THEN #PageFwRequest := #CurrentPage; END_IF;
   IF #_w1 AND "DB21_DisplayGeneralData".dbx0_4 THEN #PageFwRequest := 28; END_IF;
END_REGION

REGION Network 9: Timer 8 page selection
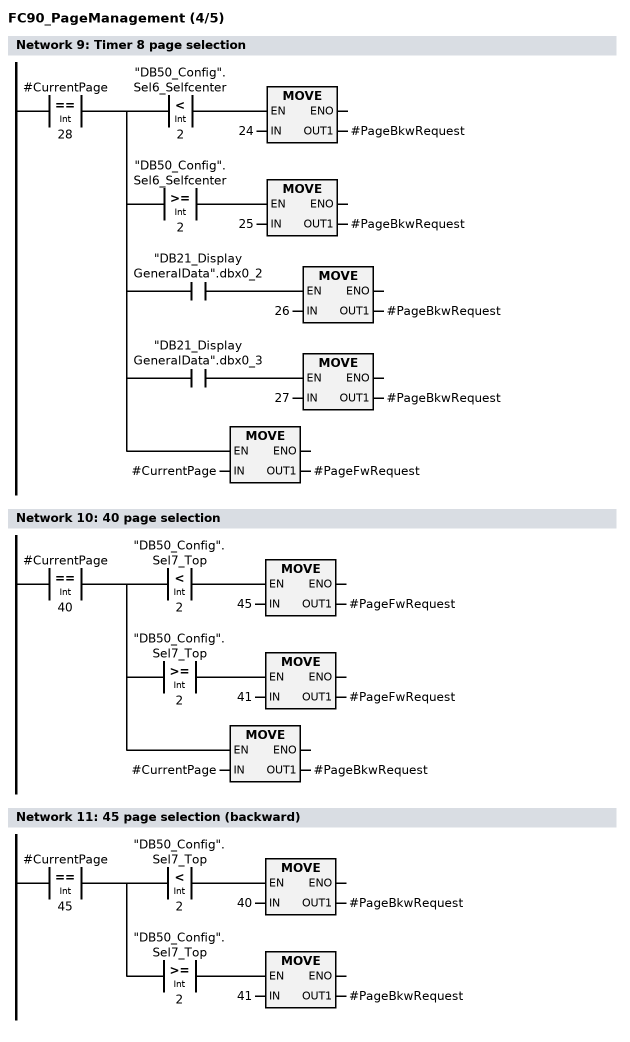
   RUNG wire#powerrail
      { S7_Templates := "SrcType := Int" } EQ_Contact(in1 := #CurrentPage, in2 := 28)
      wire#w1
      { S7_Templates := "SrcType := Int" } LT_Contact(in1 := "DB50_Config".Sel6_Selfcenter, in2 := 2)
      { S7_GenerateENO := "TRUE" } Move(in := 24, out1 => #PageBkwRequest)
   END_RUNG
   RUNG wire#w1
      { S7_Templates := "SrcType := Int" } GE_Contact(in1 := "DB50_Config".Sel6_Selfcenter, in2 := 2)
      { S7_GenerateENO := "TRUE" } Move(in := 25, out1 => #PageBkwRequest)
   END_RUNG
   RUNG wire#w1
      Contact( "DB21_DisplayGeneralData".dbx0_2 )
      { S7_GenerateENO := "TRUE" } Move(in := 26, out1 => #PageBkwRequest)
   END_RUNG
   RUNG wire#w1
      Contact( "DB21_DisplayGeneralData".dbx0_3 )
      { S7_GenerateENO := "TRUE" } Move(in := 27, out1 => #PageBkwRequest)
   END_RUNG
   RUNG wire#w1
      { S7_GenerateENO := "TRUE" } Move(in := #CurrentPage, out1 => #PageFwRequest)
   END_RUNG
   // the same network as SCL:
   #_w1 := #CurrentPage = 28;
   IF #_w1 AND ("DB50_Config".Sel6_Selfcenter < 2) THEN #PageBkwRequest := 24; END_IF;
   IF #_w1 AND ("DB50_Config".Sel6_Selfcenter >= 2) THEN #PageBkwRequest := 25; END_IF;
   IF #_w1 AND "DB21_DisplayGeneralData".dbx0_2 THEN #PageBkwRequest := 26; END_IF;
   IF #_w1 AND "DB21_DisplayGeneralData".dbx0_3 THEN #PageBkwRequest := 27; END_IF;
   IF #_w1 THEN #PageFwRequest := #CurrentPage; END_IF;
END_REGION

REGION Network 10: 40 page selection
   RUNG wire#powerrail
      { S7_Templates := "SrcType := Int" } EQ_Contact(in1 := #CurrentPage, in2 := 40)
      wire#w1
      { S7_Templates := "SrcType := Int" } LT_Contact(in1 := "DB50_Config".Sel7_Top, in2 := 2)
      { S7_GenerateENO := "TRUE" } Move(in := 45, out1 => #PageFwRequest)
   END_RUNG
   RUNG wire#w1
      { S7_Templates := "SrcType := Int" } GE_Contact(in1 := "DB50_Config".Sel7_Top, in2 := 2)
      { S7_GenerateENO := "TRUE" } Move(in := 41, out1 => #PageFwRequest)
   END_RUNG
   RUNG wire#w1
      { S7_GenerateENO := "TRUE" } Move(in := #CurrentPage, out1 => #PageBkwRequest)
   END_RUNG
   // the same network as SCL:
   #_w1 := #CurrentPage = 40;
   IF #_w1 AND ("DB50_Config".Sel7_Top < 2) THEN #PageFwRequest := 45; END_IF;
   IF #_w1 AND ("DB50_Config".Sel7_Top >= 2) THEN #PageFwRequest := 41; END_IF;
   IF #_w1 THEN #PageBkwRequest := #CurrentPage; END_IF;
END_REGION

REGION Network 11: 45 page selection (backward)
   RUNG wire#powerrail
      { S7_Templates := "SrcType := Int" } EQ_Contact(in1 := #CurrentPage, in2 := 45)
      wire#w1
      { S7_Templates := "SrcType := Int" } LT_Contact(in1 := "DB50_Config".Sel7_Top, in2 := 2)
      { S7_GenerateENO := "TRUE" } Move(in := 40, out1 => #PageBkwRequest)
   END_RUNG
   RUNG wire#w1
      { S7_Templates := "SrcType := Int" } GE_Contact(in1 := "DB50_Config".Sel7_Top, in2 := 2)
      { S7_GenerateENO := "TRUE" } Move(in := 41, out1 => #PageBkwRequest)
   END_RUNG
   // the same network as SCL:
   #_w1 := #CurrentPage = 45;
   IF #_w1 AND ("DB50_Config".Sel7_Top < 2) THEN #PageBkwRequest := 40; END_IF;
   IF #_w1 AND ("DB50_Config".Sel7_Top >= 2) THEN #PageBkwRequest := 41; END_IF;
END_REGION

REGION Network 12
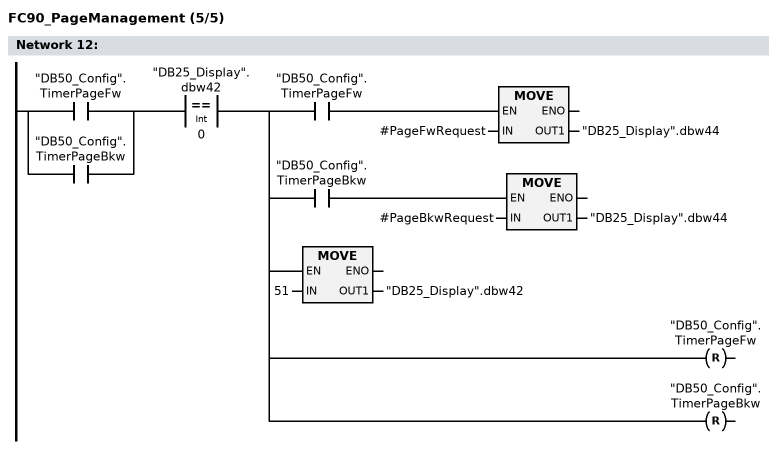
   RUNG wire#powerrail
      Contact( "DB50_Config".TimerPageFw )
      wire#w1
      { S7_Templates := "SrcType := Int" } EQ_Contact(in1 := "DB25_Display".dbw42, in2 := 0)
      wire#w2
      Contact( "DB50_Config".TimerPageFw )
      { S7_GenerateENO := "TRUE" } Move(in := #PageFwRequest, out1 => "DB25_Display".dbw44)
   END_RUNG
   RUNG wire#powerrail
      Contact( "DB50_Config".TimerPageBkw )
   END_RUNG wire#w1
   RUNG wire#w2
      Contact( "DB50_Config".TimerPageBkw )
      { S7_GenerateENO := "TRUE" } Move(in := #PageBkwRequest, out1 => "DB25_Display".dbw44)
   END_RUNG
   RUNG wire#w2
      { S7_GenerateENO := "TRUE" } Move(in := 51, out1 => "DB25_Display".dbw42)
   END_RUNG
   RUNG wire#w2
      R_Coil( "DB50_Config".TimerPageFw )
   END_RUNG
   RUNG wire#w2
      R_Coil( "DB50_Config".TimerPageBkw )
   END_RUNG
   // the same network as SCL:
   #_w1 := ("DB50_Config".TimerPageFw OR "DB50_Config".TimerPageBkw) AND ("DB25_Display".dbw42 = 0);
   IF #_w1 AND "DB50_Config".TimerPageFw THEN "DB25_Display".dbw44 := #PageFwRequest; END_IF;
   IF #_w1 AND "DB50_Config".TimerPageBkw THEN "DB25_Display".dbw44 := #PageBkwRequest; END_IF;
   IF #_w1 THEN
       "DB25_Display".dbw42 := 51;
       "DB50_Config".TimerPageFw := FALSE;
       "DB50_Config".TimerPageBkw := FALSE;
   END_IF;
END_REGION
END_FUNCTION

FUNCTION "Normalisation" : Void   // FC15, FBD
{ S7_Optimized_Access := 'TRUE' }
VERSION : 0.1
// stored: AutoNumber true, IsIECCheckEnabled false, SetENOAutomatically false, UDAEnableTagReadback false
   VAR_INPUT
      value_REAL : Real;
      normalisation : Real;
   END_VAR
   VAR_OUTPUT
      value_INT : Int;
   END_VAR
   VAR_TEMP
      temp_value_DINT : DInt;
      temp_value_REAL : Real;
   END_VAR
BEGIN

REGION Network 1
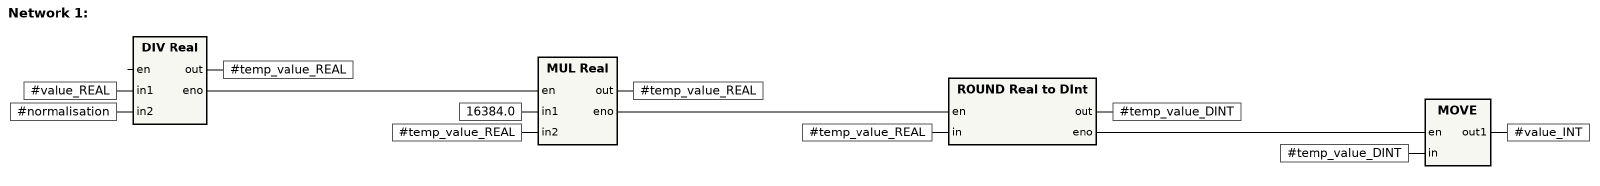
   // ENO of a box is taken as its EN; it also drops when the box reports an error
   #temp_value_REAL := #value_REAL / #normalisation;
   #temp_value_REAL := 16384.0 * #temp_value_REAL;
   #temp_value_DINT := ROUND(#temp_value_REAL);
   #value_INT := #temp_value_DINT;
END_REGION
END_FUNCTION

FUNCTION "Centrador_Paletes" : Void   // FC17, LAD
{ S7_Optimized_Access := 'TRUE' }
VERSION : 0.1
// stored: AutoNumber true, IsIECCheckEnabled false, SetENOAutomatically false, UDAEnableTagReadback false
   VAR_TEMP
      Detetor_Palete : Bool;
      Comando_Tapete_Centrador : Bool;
      Start : Bool;
      Setpoint : Real;
      ActVelocity : Real;
      RefSpeed : Real;
   END_VAR
   VAR_TEMP   // added for the SCL form of the ladder/FBD networks
      _w1 : Bool;
   END_VAR
BEGIN

REGION Network 1: Motor tapete de rolos do centrador
   // Tapete só anda se ambas as barras centradoras estiverem na posição aberta e pára quando deteta palete
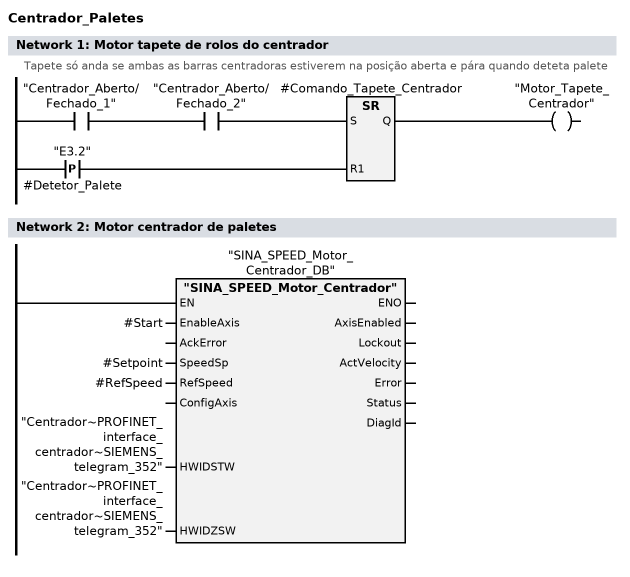
   RUNG wire#powerrail
      Contact( "Centrador_Aberto/Fechado_1" )
      Contact( "Centrador_Aberto/Fechado_2" )
      S_SR(operand := #Comando_Tapete_Centrador, r1 := wire#w1)
      Coil( "Motor_Tapete_Centrador" )
   END_RUNG
   RUNG wire#powerrail
      P_Contact(operand := "E3.2", bit := #Detetor_Palete)
   END_RUNG wire#w1
   // the same network as SCL:
   #_w1 := "E3.2" AND NOT #Detetor_Palete;   // rising edge of "E3.2"
   #Detetor_Palete := "E3.2";
   IF "Centrador_Aberto/Fechado_1" AND "Centrador_Aberto/Fechado_2" THEN
       #Comando_Tapete_Centrador := TRUE;   // SR flip-flop
   END_IF;
   IF #_w1 THEN #Comando_Tapete_Centrador := FALSE; END_IF;
   "Motor_Tapete_Centrador" := #Comando_Tapete_Centrador;
END_REGION

REGION Network 2: Motor centrador de paletes
   RUNG wire#powerrail
      "SINA_SPEED_Motor_Centrador_DB"(EnableAxis := #Start, AckError :=, SpeedSp := #Setpoint, RefSpeed := #RefSpeed, ConfigAxis :=, HWIDSTW := "Centrador~PROFINET_interface_centrador~SIEMENS_telegram_352", HWIDZSW := "Centrador~PROFINET_interface_centrador~SIEMENS_telegram_352", AxisEnabled =>, Lockout =>, ActVelocity =>, Error =>, Status =>, DiagId =>)
   END_RUNG
   // the same network as SCL:
   "SINA_SPEED_Motor_Centrador_DB"(EnableAxis := #Start,   // "SINA_SPEED_Motor_Centrador"
                           SpeedSp := #Setpoint,
                           RefSpeed := #RefSpeed,
                           HWIDSTW := "Centrador~PROFINET_interface_centrador~SIEMENS_telegram_352",
                           HWIDZSW := "Centrador~PROFINET_interface_centrador~SIEMENS_telegram_352");
END_REGION
END_FUNCTION

FUNCTION_BLOCK "SINA_SPEED_Motor_Centrador"
TITLE = 'Speed Control with SINAMICS and S7'
{ S7_Optimized_Access := 'TRUE' }
AUTHOR : DRVDPS7
FAMILY : DRIVES
NAME : SINA_SPD
VERSION : 5.1
//Copyright (C) Siemens AG 2012. All Rights Reserved. Confidential
//-------------------------------------------------------------------------------------- 
//SINA_SPEED: Drehzahlregelung mit dem Antriebsbaustein SINAMICS S120/G120 <-> S7-1200
//------------------------------------------------------------------------------------- Ersteller: Siemens AG Erlangen A&D MC PM   Datum:  07.07.10        Vers.:2.1
//Änderung:  J.B. Typical Team                       07.12.12              2.2
//    Umsetzung in SCL / TIA 
//Änderung:  J.B. Typical Team                       29.04.13              2.3
//    1. "Q" an den AusgÃ¤nge entfernen
//    2. Neuer Ausgang PwrInhibit
//Änderung:  J.B. Typical Team                       28.06.13              2.4
//    Ã„nderung HW-Zugriff Ã¼ber LOG2MOD
//     
//Änderung:  J.B. Typical Team                       18.07.13              2.5
//    Ã„nderung HW-Zugriff Ã¼ber zwei HW-EingÃ¤nge
//
//Änderung:  J.B. Typical Team                       17.07.14              3.0
//    Optimmierung
//
//Änderung:  J.B. Typical Team                       30.07.14              4.0
//    Festlegung auf einheitlicher neuer Version 4.0
//
//Änderung:  P.Z. Typical Team                       03.12.15              4.1
//    Schnittstelle an Programmierleitfadeb TIA-Potal angepasst
//    zusÃ¤tzlicher Eingang "ConfigAxis" fÃ¼r STW-Bits
//
//Änderung:  G.F. Typical Team                       01.03.16              4.2
//    Sollwert auf INT - Grenzen begrenzt
//Änderung:  F.G. Typical Team                       13.09.16              4.3
//    Ausgabewerte am Ausgang "Status" angepasst 
//
//Änderung:  G.F. Typical Team                       11.01.17              5.0
//    - Festlegung auf einheitlicher neuer Version 5.0 
//
//Änderung:  G.F. Typical Team                       03.05.18              5.1
//    - Alle Bits des Eingang ConfigAxis auf STW1 aufgelegt 
//
//Bibliothek V7
//Funktion: Drehzahlregelung mit dem Antriebsbaustein SINAMICS S120/G120 <-> S7-1200
//********************************************************************************************************************************************************
//************************************************************************FB283***************************************************************************
//********************************************************************************************************************************************************
   VAR_INPUT 
      EnableAxis : Bool := 0;   // 0-->1; 1 = Enable the drive (OFF2 / OFF 3 are 1 in default status) (OFF1 = 0-->1)
      AckError : Bool := 0;   // 1 = Acknowledge drive error
      SpeedSp : Real := 0.0;   // Speed standardises with the standardisation factor
      RefSpeed : Real := 0.0;   // Standardisation factor of speed
      ConfigAxis : Word := 16#003F;   // binary programmed input to control all functions in the telegram without its own function block input
      HWIDSTW : HW_IO := 0;   // Hardware Identifer set point slot
      HWIDZSW : HW_IO := 0;   // Hardware Identifer actual value slot
   END_VAR

   VAR_OUTPUT 
      AxisEnabled : Bool := 0;   // 1 = Drive is enabled
      Lockout : Bool := 0;   // 1 = Drive lockout active
      ActVelocity : Real := 0.0;   // Actual in [U/min]
      Error : Bool := 0;   // 1 = Error  (FB and Infeed)
      Status : Word := 0;   // Status output (7002 = FB in operation; 8xxx = error description  - read the manual)
      DiagId : Word := 16#0000;   // Error codes of the cyclic system funtion blocks DPWR / DPRD_DAT
   END_VAR

   VAR 
      sxSendBuf : Struct   // Send buffer
         STW1 : Word := WORD#16#0000;   // STW1sxSTW1     : STRUCT            Bit08       : BOOL:=False;              // ST-Wort-1 Bit 08 --> Reserve            Bit09       : BOOL:=False;              // ST-Wort-1 Bit 09 --> Reserve            Bit10       : BOOL:=True;               // ST-Wort-1 Bit 10 --> FÃ¼hrung durch PLC            Dir         : BOOL:=False;              // ST-Wort-1 Bit 11 --> Direction            Bit12       : BOOL:=False;              // ST-Wort-1 Bit 12 --> Haltebremse unbedingt Ã¶ffnen            Bit13       : BOOL:=False;              // ST-Wort-1 Bit 13 --> Motorpotenziometer Sollwert hÃ¶her            Bit14       : BOOL:=False;              // ST-Wort-1 Bit 14 --> Motorpotenziometer Sollwert tiefer            Bit15       : BOOL:=False;              // ST-Wort-1 Bit 15 --> Reserviert            Off1        : BOOL:=False;              // ST-Wort-1 Bit 00 --> OFF1/ON (flanks acceptance)            Off2        : BOOL:=True;               // ST-Wort-1 Bit 01 --> OFF2/ON (enable possible)            Off3        : BOOL:=True;               // ST-Wort-1 Bit 02 --> OFF3/ON (enable possible)            InvEn       : BOOL:=True;               // ST-Wort-1 Bit 03 --> Enable controller            RampEn      : BOOL:=True;               // ST-Wort-1 Bit 04 --> Ramp enable            RampOn      : BOOL:=True;               // ST-Wort-1 Bit 05 --> Ramp On            SpEn        : BOOL:=True;               // ST-Wort-1 Bit 06 --> Speed set point enable            AckFlt      : BOOL:=False;              // ST-Wort-1 Bit 07 --> Acknowledge fault         END_STRUCT;
         Velocity : Word := WORD#16#0000;   // Setpoint of velocity
      END_STRUCT;
      sxRecvBuf : Struct   // Receive buffer
         ZSW1 : Word := WORD#16#0000;   // ZSW1sxZSW1     : STRUCT            SpDev       : BOOL:=False;              // ZSW-Wort-1 = Schleppfehler im Toleranzbereich            Pcd         : BOOL:=False;              // ZSW-Wort-1 = PZD-FÃ¼hrung erreicht            Comp        : BOOL:=False;              // ZSW-Wort-1 = Zielposition erreicht            CurLim      : BOOL:=False;              // ZSW-Wort-1 = Referenzpunkt gesetzt            Brake       : BOOL:=False;              // ZSW-Wort-1 = Haltebremse Ã¶ffnen            Motover     : BOOL:=False;              // ZSW-Wort-1 = keine Warnung Ãœbertemperatur Motor            Dir         : BOOL:=False;              // ZSW-Wort-1 = Direction            Invover     : BOOL:=False;              // ZSW-Wort-1 = keine Warnung thermische Ãœberlast Leistungsteil            Rts         : BOOL:=False;              // ZSW-Wort-1 = Ready to power up / to start            Rdy         : BOOL:=False;              // ZSW-Wort-1 = Ready to operate            IOp         : BOOL:=False;              // ZSW-Wort-1 = In operation (operation enabled)            Fault       : BOOL:=False;              // ZSW-Wort-1 = Fault present            NoOff2      : BOOL:=False;              // ZSW-Wort-1 = OFF2 inactive            NoOff3      : BOOL:=False;              // ZSW-Wort-1 = OFF3 inactive            Inhibit     : BOOL:=False;              // ZSW-Wort-1 = Power ON inhibit active             Alarm       : BOOL:=False;              // ZSW-Wort-1 = Alarm / Warning present                     END_STRUCT;
         Velocity : Word := WORD#16#0000;   // Feedback of velocity
      END_STRUCT;
   END_VAR

   VAR_TEMP 
      piRetSFC : Int;   // Status for fault analysis
      piCount : Int;   // Freely available counter variable 3
      prVelocity : Real;   // velocity
      pdRecvBuf : DWord;   // Buffer of Recv-Value
      pdSendBuf : DWord;   // Buffer of Send-Value
      phLAddr : HW_IO;   // Start addr from the I/O process image area of mod (DEC) for DPWR_DAT/DPRD_DAT
      swSendBuf : Array[0..1] of Word;   // Sendepuffer
      swRecvBuf : Array[0..1] of Word;   // Empfangspuffer         Static variables
   END_VAR


BEGIN
	
	//=============================================================================
	//SIEMENS AG
	//(c)Copyright 2017 All Rights Reserved
	//-----------------------------------------------------------------------------
	// Library: DriveLib
	// Tested with: S7-1516-3 PN/DP V1.8
	// Engineering: TIA Portal V14
	// Restrictions: -
	// Requirements: S7-1200 / S7-1500
	// Functionality: cyclic communication between a SINAMICS a PLC.
	//                If in HWConfig Std.TLG 1 is projected 2 PZD-words are exchanged
	//                in every bus cycle.
	//                The parametrisation of these words is described in the manual of the
	//                SINAMICS
	//=============================================================================
	
	// Schreibdaten zusammenstellen
	// Steuerword aufbereiten
	
	#sxSendBuf.STW1.%X0 := #EnableAxis;
	#sxSendBuf.STW1.%X1 := #ConfigAxis.%X0;
	#sxSendBuf.STW1.%X2 := #ConfigAxis.%X1;
	#sxSendBuf.STW1.%X3 := #ConfigAxis.%X2;
	#sxSendBuf.STW1.%X4 := #ConfigAxis.%X3;
	#sxSendBuf.STW1.%X5 := #ConfigAxis.%X4;
	#sxSendBuf.STW1.%X6 := #ConfigAxis.%X5;
	#sxSendBuf.STW1.%X7 := #AckError;
	#sxSendBuf.STW1.%X8 := #ConfigAxis.%X10;
	#sxSendBuf.STW1.%X9 := #ConfigAxis.%X11;
	#sxSendBuf.STW1.%X10 := TRUE;
	#sxSendBuf.STW1.%X11 := #ConfigAxis.%X6;
	#sxSendBuf.STW1.%X12 := #ConfigAxis.%X7;
	#sxSendBuf.STW1.%X13 := #ConfigAxis.%X8;
	#sxSendBuf.STW1.%X14 := #ConfigAxis.%X9;
	#sxSendBuf.STW1.%X15 := #ConfigAxis.%X12;
	
	// Geschwindigkeit
	IF #RefSpeed <> 0 THEN
	  #prVelocity := #SpeedSp * (16384.0 / #RefSpeed);
	  // Limit REAL - Variable to INT - Limits
	  IF #prVelocity > 32767 THEN
	    #prVelocity := 32767;
	  ELSIF #prVelocity < -32768 THEN
	    #prVelocity := -32768;
	  ELSE
	    ; // not needed
	  END_IF;
	  #sxSendBuf.Velocity := INT_TO_WORD(REAL_TO_INT(#prVelocity));
	  
	ELSE
	  #sxSendBuf.Velocity := W#16#0;
	END_IF;
	#swSendBuf[0] := #sxSendBuf.STW1;
	#swSendBuf[1] := #sxSendBuf.Velocity;
	
	//Prozessdaten zur Signalbaugruppe schreiben
	#piRetSFC := DPWR_DAT(LADDR := #HWIDSTW,
	                      RECORD := #swSendBuf);
	
	// Fehler der RÃ¼ckmeldung ausgeben
	#DiagId := INT_TO_WORD(#piRetSFC);
	
	//kein Fehler beim Schreiben
	IF #piRetSFC = 0 THEN
	  
	  //kein Fehler beim Schreiben
	  IF #piRetSFC = 0 THEN
	    
	    //Prozessdaten von der Signalbaugruppe lesen
	    #piRetSFC := DPRD_DAT(LADDR := #HWIDZSW,
	                          RECORD => #swRecvBuf);
	    
	    // Fehler der RÃ¼ckmeldung ausgeben
	    #DiagId := INT_TO_WORD(#piRetSFC);
	  END_IF;
	  
	  //Fehler beim Lesen (Profibus-Kommunikation unterbrochen)
	  IF #piRetSFC <> 0 THEN
	    
	    // Fehler
	    #Error := TRUE;
	    #Status := 16#8600;
	    
	    // Zustandsworte lÃ¶schen
	    #sxRecvBuf.ZSW1.%X8 := 0;
	    #sxRecvBuf.ZSW1.%X9 := 0;
	    #sxRecvBuf.ZSW1.%X10 := 0;
	    #sxRecvBuf.ZSW1.%X11 := 0;
	    #sxRecvBuf.ZSW1.%X12 := 0;
	    #sxRecvBuf.ZSW1.%X13 := 0;
	    #sxRecvBuf.ZSW1.%X14 := 0;
	    #sxRecvBuf.ZSW1.%X15 := 0;
	    #sxRecvBuf.ZSW1.%X0 := 0;
	    #sxRecvBuf.ZSW1.%X1 := 0;
	    #sxRecvBuf.ZSW1.%X2 := 0;
	    #sxRecvBuf.ZSW1.%X3 := 0;
	    #sxRecvBuf.ZSW1.%X4 := 0;
	    #sxRecvBuf.ZSW1.%X5 := 0;
	    #sxRecvBuf.ZSW1.%X6 := 0;
	    #sxRecvBuf.ZSW1.%X7 := 0;
	    
	    
	    (*#sxRecvBuf.sxZSW1.SpDev   := 0;
	    #sxRecvBuf.sxZSW1.Pcd     := 0;
	    #sxRecvBuf.sxZSW1.Comp    := 0;
	    #sxRecvBuf.sxZSW1.CurLim  := 0;
	    #sxRecvBuf.sxZSW1.Brake   := 0;
	    #sxRecvBuf.sxZSW1.Motover := 0;
	    #sxRecvBuf.sxZSW1.Dir     := 0;
	    #sxRecvBuf.sxZSW1.Invover := 0;
	    #sxRecvBuf.sxZSW1.Rts     := 0;
	    #sxRecvBuf.sxZSW1.Rdy     := 0;
	    #sxRecvBuf.sxZSW1.IOp     := 0;
	    #sxRecvBuf.sxZSW1.Fault   := 0;
	    #sxRecvBuf.sxZSW1.NoOff2  := 0;
	    #sxRecvBuf.sxZSW1.NoOff3  := 0;
	    #sxRecvBuf.sxZSW1.Inhibit := 0;
	    #sxRecvBuf.sxZSW1.Alarm   := 0;*)
	    
	    #sxRecvBuf.Velocity := W#16#00;
	    
	    // Werte auslesen
	  ELSE
	    #sxRecvBuf.ZSW1 := #swRecvBuf[0];
	    #sxRecvBuf.Velocity := #swRecvBuf[1];
	    
	    // ZSW1 aufbereiten                       
	    #AxisEnabled := #sxRecvBuf.ZSW1.%X2;
	    #Error := #sxRecvBuf.ZSW1.%X3 OR #sxRecvBuf.ZSW1.%X6;
	    #Lockout := #sxRecvBuf.ZSW1.%X6;
	    
	    // Fehler auswerten
	    IF #sxRecvBuf.ZSW1.%X3 THEN
	      #Status := 16#8401;
	    ELSIF #sxRecvBuf.ZSW1.%X6 THEN
	      #Status := 16#8402;
	    ELSE
	      #Status := 16#7002;
	    END_IF;
	    
	    (*#Busy       := #sxRecvBuf.sxZSW1.IOp;
	    #Error      := #sxRecvBuf.sxZSW1.Fault OR #sxRecvBuf.sxZSW1.Inhibit;
	    #PwrInhibit := #sxRecvBuf.sxZSW1.Inhibit;            
	
	    // Fehler auswerten
	    IF #sxRecvBuf.sxZSW1.Fault THEN
	        #ErrorId := 1;
	    ELSIF #sxRecvBuf.sxZSW1.Inhibit THEN 
	        #ErrorId := 2;
	    ELSE
	        #ErrorId := 0;    
	    END_IF;*)
	    
	    // Geschwindigkeit
	    IF #RefSpeed <> 0 THEN
	      #ActVelocity := INT_TO_REAL(WORD_TO_INT(#sxRecvBuf.Velocity)) / (16384.0 / #RefSpeed);
	    ELSE
	      #ActVelocity := 0.0;
	    END_IF;
	  END_IF;
	ELSE
	  
	  // Fehler
	  #Error := TRUE;
	  #Status := 16#8601;
	  
	END_IF;
	
	
	
END_FUNCTION_BLOCK

FUNCTION "FC00_SupportIn" : Void   // FC0, LAD
TITLE = Input support memory
{ S7_Optimized_Access := 'FALSE' }
AUTHOR : Robopac
VERSION : 0.0
// stored: AutoNumber false, IsIECCheckEnabled false, SetENOAutomatically false, UDAEnableTagReadback false
   VAR_TEMP
      AC1 : Int;
      AC2 : Int;
   END_VAR
BEGIN

REGION Network 1: STANDARD
END_REGION

REGION Network 2: Pressure switch (Technoplat)
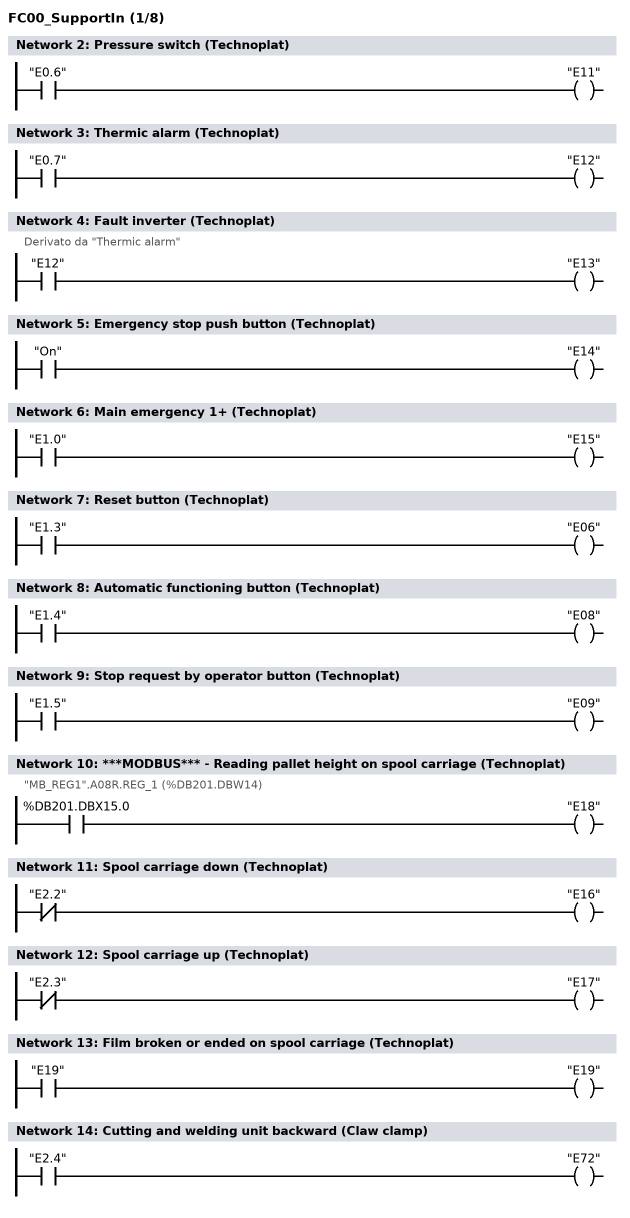
   RUNG wire#powerrail
      Contact( "E0.6" )
      Coil( "E11" )
   END_RUNG
   // the same network as SCL:
   "E11" := "E0.6";
END_REGION

REGION Network 3: Thermic alarm (Technoplat)
   RUNG wire#powerrail
      Contact( "E0.7" )
      Coil( "E12" )
   END_RUNG
   // the same network as SCL:
   "E12" := "E0.7";
END_REGION

REGION Network 4: Fault inverter (Technoplat)
   // Derivato da "Thermic alarm"
   RUNG wire#powerrail
      Contact( "E12" )
      Coil( "E13" )
   END_RUNG
   // the same network as SCL:
   "E13" := "E12";
END_REGION

REGION Network 5: Emergency stop push button (Technoplat)
   RUNG wire#powerrail
      Contact( "On" )
      Coil( "E14" )
   END_RUNG
   // the same network as SCL:
   "E14" := "On";
END_REGION

REGION Network 6: Main emergency 1+ (Technoplat)
   RUNG wire#powerrail
      Contact( "E1.0" )
      Coil( "E15" )
   END_RUNG
   // the same network as SCL:
   "E15" := "E1.0";
END_REGION

REGION Network 7: Reset button (Technoplat)
   RUNG wire#powerrail
      Contact( "E1.3" )
      Coil( "E06" )
   END_RUNG
   // the same network as SCL:
   "E06" := "E1.3";
END_REGION

REGION Network 8: Automatic functioning button (Technoplat)
   RUNG wire#powerrail
      Contact( "E1.4" )
      Coil( "E08" )
   END_RUNG
   // the same network as SCL:
   "E08" := "E1.4";
END_REGION

REGION Network 9: Stop request by operator button (Technoplat)
   RUNG wire#powerrail
      Contact( "E1.5" )
      Coil( "E09" )
   END_RUNG
   // the same network as SCL:
   "E09" := "E1.5";
END_REGION

REGION Network 10: ***MODBUS*** - Reading pallet height on spool carriage (Technoplat)
   // "MB_REG1".A08R.REG_1 (%DB201.DBW14)
   RUNG wire#powerrail
      Contact( %DB201.DBX15.0 )
      Coil( "E18" )
   END_RUNG
   // the same network as SCL:
   "E18" := %DB201.DBX15.0;
END_REGION

REGION Network 11: Spool carriage down (Technoplat)
   RUNG wire#powerrail
      I_Contact( "E2.2" )
      Coil( "E16" )
   END_RUNG
   // the same network as SCL:
   "E16" := NOT "E2.2";
END_REGION

REGION Network 12: Spool carriage up (Technoplat)
   RUNG wire#powerrail
      I_Contact( "E2.3" )
      Coil( "E17" )
   END_RUNG
   // the same network as SCL:
   "E17" := NOT "E2.3";
END_REGION

REGION Network 13: Film broken or ended on spool carriage (Technoplat)
   RUNG wire#powerrail
      Contact( "E19" )
      Coil( "E19" )
   END_RUNG
   // the same network as SCL:
   "E19" := "E19";
END_REGION

REGION Network 14: Cutting and welding unit backward (Claw clamp)
   RUNG wire#powerrail
      Contact( "E2.4" )
      Coil( "E72" )
   END_RUNG
   // the same network as SCL:
   "E72" := "E2.4";
END_REGION

REGION Network 15: Cutting and welding unit forward (Claw clamp)
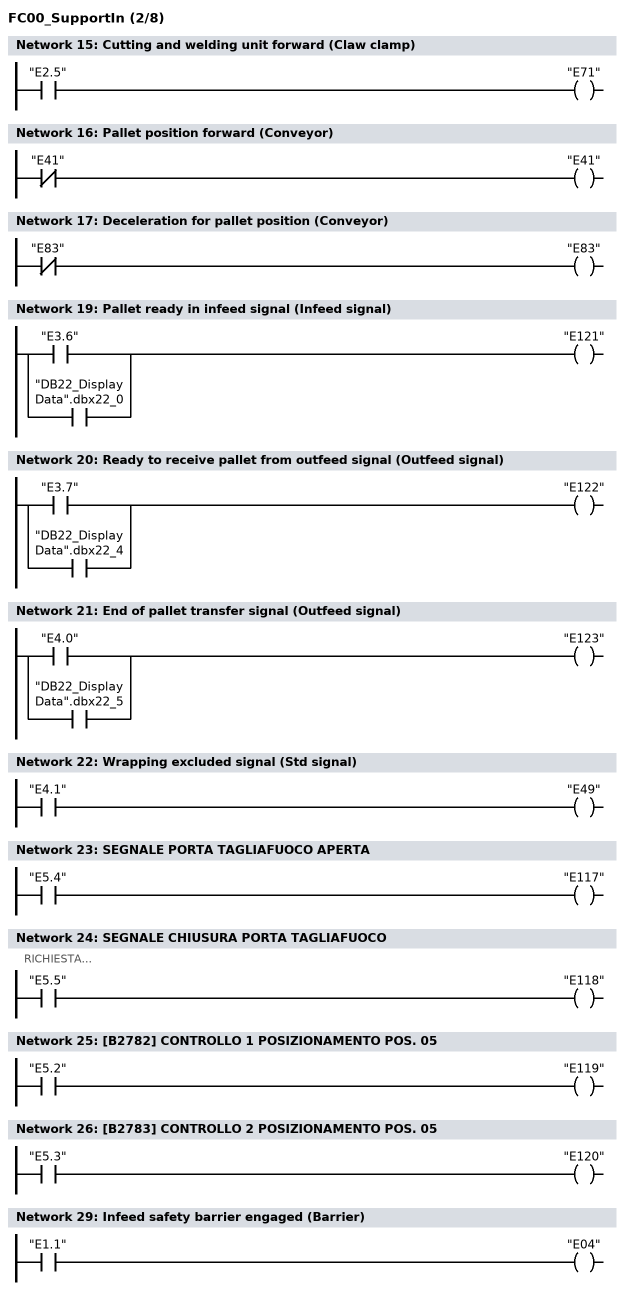
   RUNG wire#powerrail
      Contact( "E2.5" )
      Coil( "E71" )
   END_RUNG
   // the same network as SCL:
   "E71" := "E2.5";
END_REGION

REGION Network 16: Pallet position forward (Conveyor)
   RUNG wire#powerrail
      I_Contact( "E41" )
      Coil( "E41" )
   END_RUNG
   // the same network as SCL:
   "E41" := NOT "E41";
END_REGION

REGION Network 17: Deceleration for pallet position (Conveyor)
   RUNG wire#powerrail
      I_Contact( "E83" )
      Coil( "E83" )
   END_RUNG
   // the same network as SCL:
   "E83" := NOT "E83";
END_REGION

REGION Network 18: EXCHANGE SIGNALS
END_REGION

REGION Network 19: Pallet ready in infeed signal (Infeed signal)
   RUNG wire#powerrail
      Contact( "E3.6" )
      wire#w1
      Coil( "E121" )
   END_RUNG
   RUNG wire#powerrail
      Contact( "DB22_DisplayData".dbx22_0 )
   END_RUNG wire#w1
   // the same network as SCL:
   "E121" := "E3.6" OR "DB22_DisplayData".dbx22_0;
END_REGION

REGION Network 20: Ready to receive pallet from outfeed signal (Outfeed signal)
   RUNG wire#powerrail
      Contact( "E3.7" )
      wire#w1
      Coil( "E122" )
   END_RUNG
   RUNG wire#powerrail
      Contact( "DB22_DisplayData".dbx22_4 )
   END_RUNG wire#w1
   // the same network as SCL:
   "E122" := "E3.7" OR "DB22_DisplayData".dbx22_4;
END_REGION

REGION Network 21: End of pallet transfer signal (Outfeed signal)
   RUNG wire#powerrail
      Contact( "E4.0" )
      wire#w1
      Coil( "E123" )
   END_RUNG
   RUNG wire#powerrail
      Contact( "DB22_DisplayData".dbx22_5 )
   END_RUNG wire#w1
   // the same network as SCL:
   "E123" := "E4.0" OR "DB22_DisplayData".dbx22_5;
END_REGION

REGION Network 22: Wrapping excluded signal (Std signal)
   RUNG wire#powerrail
      Contact( "E4.1" )
      Coil( "E49" )
   END_RUNG
   // the same network as SCL:
   "E49" := "E4.1";
END_REGION

REGION Network 23: SEGNALE PORTA TAGLIAFUOCO APERTA
   RUNG wire#powerrail
      Contact( "E5.4" )
      Coil( "E117" )
   END_RUNG
   // the same network as SCL:
   "E117" := "E5.4";
END_REGION

REGION Network 24: SEGNALE CHIUSURA PORTA TAGLIAFUOCO
   // RICHIESTA...
   RUNG wire#powerrail
      Contact( "E5.5" )
      Coil( "E118" )
   END_RUNG
   // the same network as SCL:
   "E118" := "E5.5";
END_REGION

REGION Network 25: [B2782] CONTROLLO 1 POSIZIONAMENTO POS. 05
   RUNG wire#powerrail
      Contact( "E5.2" )
      Coil( "E119" )
   END_RUNG
   // the same network as SCL:
   "E119" := "E5.2";
END_REGION

REGION Network 26: [B2783] CONTROLLO 2 POSIZIONAMENTO POS. 05
   RUNG wire#powerrail
      Contact( "E5.3" )
      Coil( "E120" )
   END_RUNG
   // the same network as SCL:
   "E120" := "E5.3";
END_REGION

REGION Network 27: ACCESSORIES
END_REGION

REGION Network 28: ***BARRIERS***
END_REGION

REGION Network 29: Infeed safety barrier engaged (Barrier)
   RUNG wire#powerrail
      Contact( "E1.1" )
      Coil( "E04" )
   END_RUNG
   // the same network as SCL:
   "E04" := "E1.1";
END_REGION

REGION Network 30: Outfeed safety barrier engaged (Barrier)
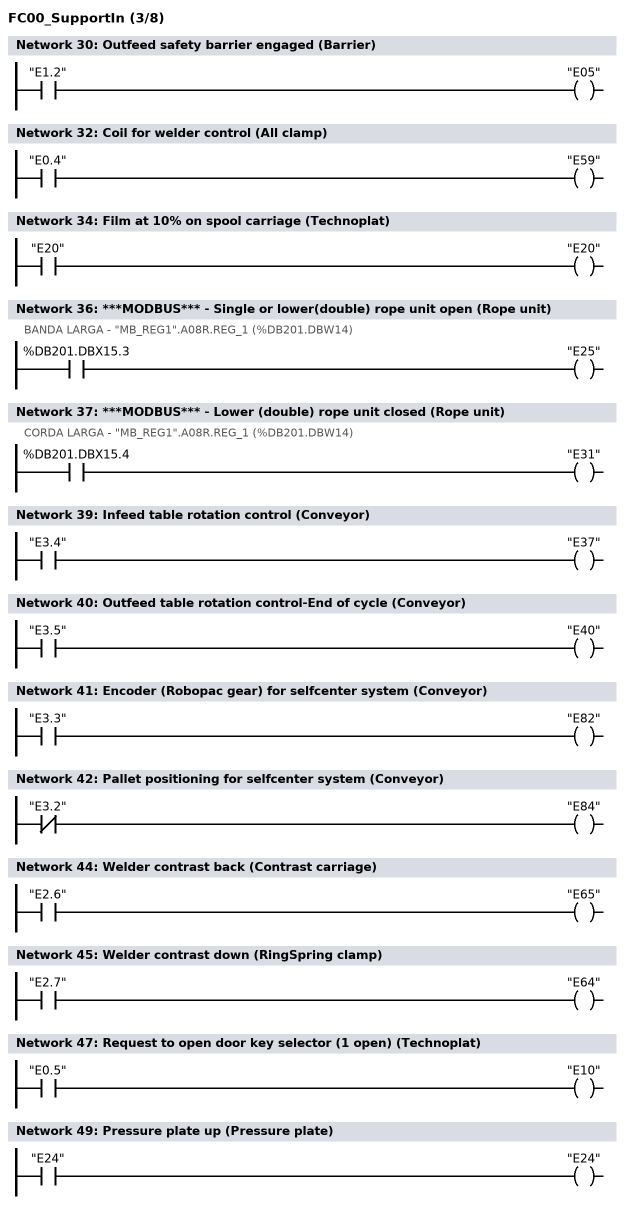
   RUNG wire#powerrail
      Contact( "E1.2" )
      Coil( "E05" )
   END_RUNG
   // the same network as SCL:
   "E05" := "E1.2";
END_REGION

REGION Network 31: ***WELDER***
END_REGION

REGION Network 32: Coil for welder control (All clamp)
   RUNG wire#powerrail
      Contact( "E0.4" )
      Coil( "E59" )
   END_RUNG
   // the same network as SCL:
   "E59" := "E0.4";
END_REGION

REGION Network 33: ***ES_FILM***
END_REGION

REGION Network 34: Film at 10% on spool carriage (Technoplat)
   RUNG wire#powerrail
      Contact( "E20" )
      Coil( "E20" )
   END_RUNG
   // the same network as SCL:
   "E20" := "E20";
END_REGION

REGION Network 35: ***BAND/ROPE***
END_REGION

REGION Network 36: ***MODBUS*** - Single or lower(double) rope unit open (Rope unit)
   // BANDA LARGA - "MB_REG1".A08R.REG_1 (%DB201.DBW14)
   RUNG wire#powerrail
      Contact( %DB201.DBX15.3 )
      Coil( "E25" )
   END_RUNG
   // the same network as SCL:
   "E25" := %DB201.DBX15.3;
END_REGION

REGION Network 37: ***MODBUS*** - Lower (double) rope unit closed (Rope unit)
   // CORDA LARGA - "MB_REG1".A08R.REG_1 (%DB201.DBW14)
   RUNG wire#powerrail
      Contact( %DB201.DBX15.4 )
      Coil( "E31" )
   END_RUNG
   // the same network as SCL:
   "E31" := %DB201.DBX15.4;
END_REGION

REGION Network 38: ***SELF-CENTER***
END_REGION

REGION Network 39: Infeed table rotation control (Conveyor)
   RUNG wire#powerrail
      Contact( "E3.4" )
      Coil( "E37" )
   END_RUNG
   // the same network as SCL:
   "E37" := "E3.4";
END_REGION

REGION Network 40: Outfeed table rotation control-End of cycle (Conveyor)
   RUNG wire#powerrail
      Contact( "E3.5" )
      Coil( "E40" )
   END_RUNG
   // the same network as SCL:
   "E40" := "E3.5";
END_REGION

REGION Network 41: Encoder (Robopac gear) for selfcenter system (Conveyor)
   RUNG wire#powerrail
      Contact( "E3.3" )
      Coil( "E82" )
   END_RUNG
   // the same network as SCL:
   "E82" := "E3.3";
END_REGION

REGION Network 42: Pallet positioning for selfcenter system (Conveyor)
   RUNG wire#powerrail
      I_Contact( "E3.2" )
      Coil( "E84" )
   END_RUNG
   // the same network as SCL:
   "E84" := NOT "E3.2";
END_REGION

REGION Network 43: ***CONTRAST***
END_REGION

REGION Network 44: Welder contrast back (Contrast carriage)
   RUNG wire#powerrail
      Contact( "E2.6" )
      Coil( "E65" )
   END_RUNG
   // the same network as SCL:
   "E65" := "E2.6";
END_REGION

REGION Network 45: Welder contrast down (RingSpring clamp)
   RUNG wire#powerrail
      Contact( "E2.7" )
      Coil( "E64" )
   END_RUNG
   // the same network as SCL:
   "E64" := "E2.7";
END_REGION

REGION Network 46: ***DOOR***
END_REGION

REGION Network 47: Request to open door key selector (1 open) (Technoplat)
   RUNG wire#powerrail
      Contact( "E0.5" )
      Coil( "E10" )
   END_RUNG
   // the same network as SCL:
   "E10" := "E0.5";
END_REGION

REGION Network 48: ***PRESSURE***
END_REGION

REGION Network 49: Pressure plate up (Pressure plate)
   RUNG wire#powerrail
      Contact( "E24" )
      Coil( "E24" )
   END_RUNG
   // the same network as SCL:
   "E24" := "E24";
END_REGION

REGION Network 50: Pressure plate positioning
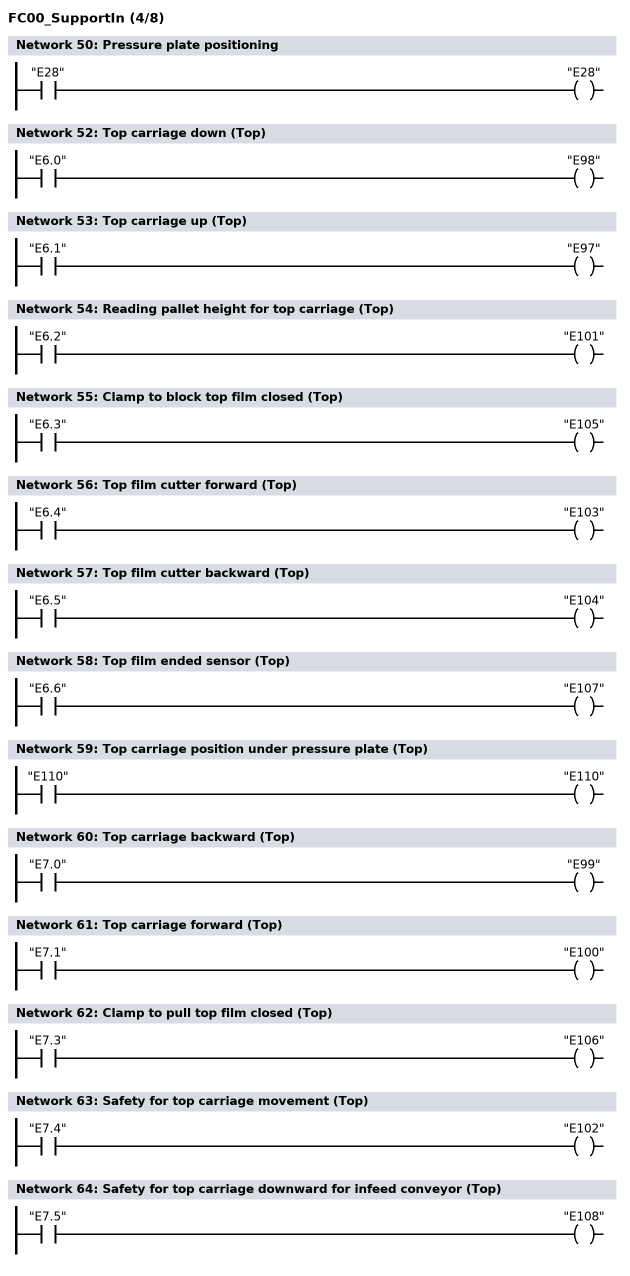
   RUNG wire#powerrail
      Contact( "E28" )
      Coil( "E28" )
   END_RUNG
   // the same network as SCL:
   "E28" := "E28";
END_REGION

REGION Network 51: ***TOP***
END_REGION

REGION Network 52: Top carriage down (Top)
   RUNG wire#powerrail
      Contact( "E6.0" )
      Coil( "E98" )
   END_RUNG
   // the same network as SCL:
   "E98" := "E6.0";
END_REGION

REGION Network 53: Top carriage up (Top)
   RUNG wire#powerrail
      Contact( "E6.1" )
      Coil( "E97" )
   END_RUNG
   // the same network as SCL:
   "E97" := "E6.1";
END_REGION

REGION Network 54: Reading pallet height for top carriage (Top)
   RUNG wire#powerrail
      Contact( "E6.2" )
      Coil( "E101" )
   END_RUNG
   // the same network as SCL:
   "E101" := "E6.2";
END_REGION

REGION Network 55: Clamp to block top film closed (Top)
   RUNG wire#powerrail
      Contact( "E6.3" )
      Coil( "E105" )
   END_RUNG
   // the same network as SCL:
   "E105" := "E6.3";
END_REGION

REGION Network 56: Top film cutter forward (Top)
   RUNG wire#powerrail
      Contact( "E6.4" )
      Coil( "E103" )
   END_RUNG
   // the same network as SCL:
   "E103" := "E6.4";
END_REGION

REGION Network 57: Top film cutter backward (Top)
   RUNG wire#powerrail
      Contact( "E6.5" )
      Coil( "E104" )
   END_RUNG
   // the same network as SCL:
   "E104" := "E6.5";
END_REGION

REGION Network 58: Top film ended sensor (Top)
   RUNG wire#powerrail
      Contact( "E6.6" )
      Coil( "E107" )
   END_RUNG
   // the same network as SCL:
   "E107" := "E6.6";
END_REGION

REGION Network 59: Top carriage position under pressure plate (Top)
   RUNG wire#powerrail
      Contact( "E110" )
      Coil( "E110" )
   END_RUNG
   // the same network as SCL:
   "E110" := "E110";
END_REGION

REGION Network 60: Top carriage backward (Top)
   RUNG wire#powerrail
      Contact( "E7.0" )
      Coil( "E99" )
   END_RUNG
   // the same network as SCL:
   "E99" := "E7.0";
END_REGION

REGION Network 61: Top carriage forward (Top)
   RUNG wire#powerrail
      Contact( "E7.1" )
      Coil( "E100" )
   END_RUNG
   // the same network as SCL:
   "E100" := "E7.1";
END_REGION

REGION Network 62: Clamp to pull top film closed (Top)
   RUNG wire#powerrail
      Contact( "E7.3" )
      Coil( "E106" )
   END_RUNG
   // the same network as SCL:
   "E106" := "E7.3";
END_REGION

REGION Network 63: Safety for top carriage movement (Top)
   RUNG wire#powerrail
      Contact( "E7.4" )
      Coil( "E102" )
   END_RUNG
   // the same network as SCL:
   "E102" := "E7.4";
END_REGION

REGION Network 64: Safety for top carriage downward for infeed conveyor (Top)
   RUNG wire#powerrail
      Contact( "E7.5" )
      Coil( "E108" )
   END_RUNG
   // the same network as SCL:
   "E108" := "E7.5";
END_REGION

REGION Network 65: Safety for top carriage downward for outfeed conveyor (Top)
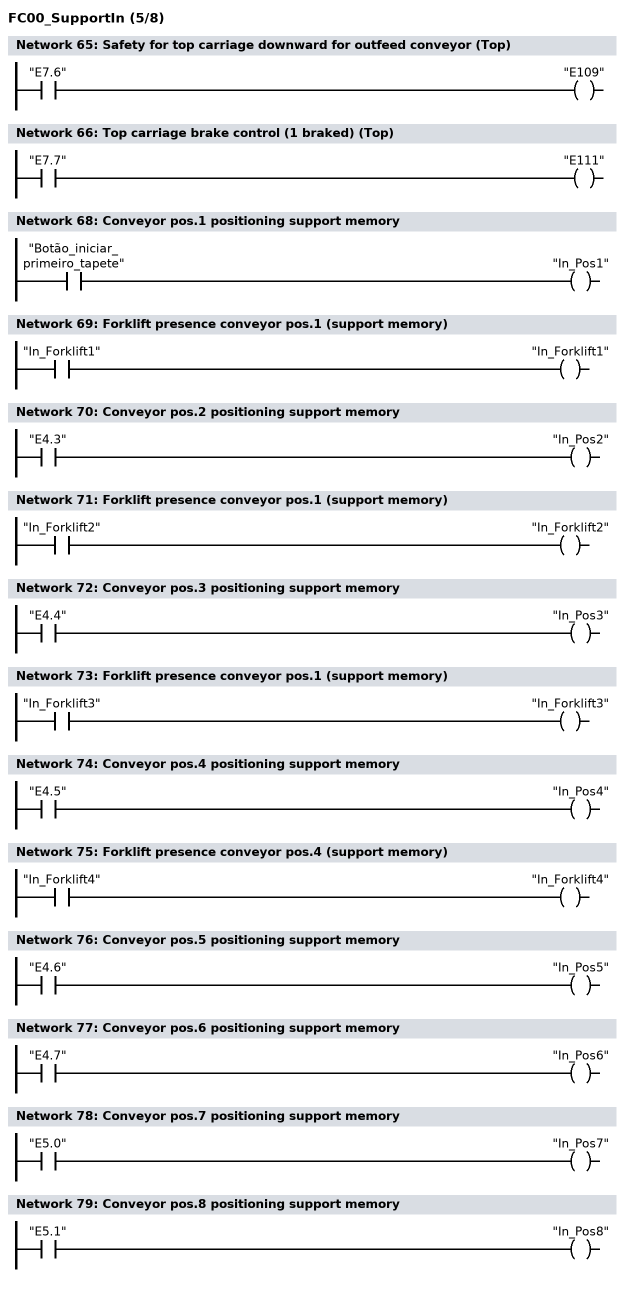
   RUNG wire#powerrail
      Contact( "E7.6" )
      Coil( "E109" )
   END_RUNG
   // the same network as SCL:
   "E109" := "E7.6";
END_REGION

REGION Network 66: Top carriage brake control (1 braked) (Top)
   RUNG wire#powerrail
      Contact( "E7.7" )
      Coil( "E111" )
   END_RUNG
   // the same network as SCL:
   "E111" := "E7.7";
END_REGION

REGION Network 67: ***CONVEYORS***
END_REGION

REGION Network 68: Conveyor pos.1 positioning support memory
   RUNG wire#powerrail
      Contact( "Botão_iniciar_primeiro_tapete" )
      Coil( "In_Pos1" )
   END_RUNG
   // the same network as SCL:
   "In_Pos1" := "Botão_iniciar_primeiro_tapete";
END_REGION

REGION Network 69: Forklift presence conveyor pos.1 (support memory)
   RUNG wire#powerrail
      Contact( "In_Forklift1" )
      Coil( "In_Forklift1" )
   END_RUNG
   // the same network as SCL:
   "In_Forklift1" := "In_Forklift1";
END_REGION

REGION Network 70: Conveyor pos.2 positioning support memory
   RUNG wire#powerrail
      Contact( "E4.3" )
      Coil( "In_Pos2" )
   END_RUNG
   // the same network as SCL:
   "In_Pos2" := "E4.3";
END_REGION

REGION Network 71: Forklift presence conveyor pos.1 (support memory)
   RUNG wire#powerrail
      Contact( "In_Forklift2" )
      Coil( "In_Forklift2" )
   END_RUNG
   // the same network as SCL:
   "In_Forklift2" := "In_Forklift2";
END_REGION

REGION Network 72: Conveyor pos.3 positioning support memory
   RUNG wire#powerrail
      Contact( "E4.4" )
      Coil( "In_Pos3" )
   END_RUNG
   // the same network as SCL:
   "In_Pos3" := "E4.4";
END_REGION

REGION Network 73: Forklift presence conveyor pos.1 (support memory)
   RUNG wire#powerrail
      Contact( "In_Forklift3" )
      Coil( "In_Forklift3" )
   END_RUNG
   // the same network as SCL:
   "In_Forklift3" := "In_Forklift3";
END_REGION

REGION Network 74: Conveyor pos.4 positioning support memory
   RUNG wire#powerrail
      Contact( "E4.5" )
      Coil( "In_Pos4" )
   END_RUNG
   // the same network as SCL:
   "In_Pos4" := "E4.5";
END_REGION

REGION Network 75: Forklift presence conveyor pos.4 (support memory)
   RUNG wire#powerrail
      Contact( "In_Forklift4" )
      Coil( "In_Forklift4" )
   END_RUNG
   // the same network as SCL:
   "In_Forklift4" := "In_Forklift4";
END_REGION

REGION Network 76: Conveyor pos.5 positioning support memory
   RUNG wire#powerrail
      Contact( "E4.6" )
      Coil( "In_Pos5" )
   END_RUNG
   // the same network as SCL:
   "In_Pos5" := "E4.6";
END_REGION

REGION Network 77: Conveyor pos.6 positioning support memory
   RUNG wire#powerrail
      Contact( "E4.7" )
      Coil( "In_Pos6" )
   END_RUNG
   // the same network as SCL:
   "In_Pos6" := "E4.7";
END_REGION

REGION Network 78: Conveyor pos.7 positioning support memory
   RUNG wire#powerrail
      Contact( "E5.0" )
      Coil( "In_Pos7" )
   END_RUNG
   // the same network as SCL:
   "In_Pos7" := "E5.0";
END_REGION

REGION Network 79: Conveyor pos.8 positioning support memory
   RUNG wire#powerrail
      Contact( "E5.1" )
      Coil( "In_Pos8" )
   END_RUNG
   // the same network as SCL:
   "In_Pos8" := "E5.1";
END_REGION

REGION Network 80: OTHER
END_REGION

REGION Network 81: Table rotation phase sensor (Technoplat)
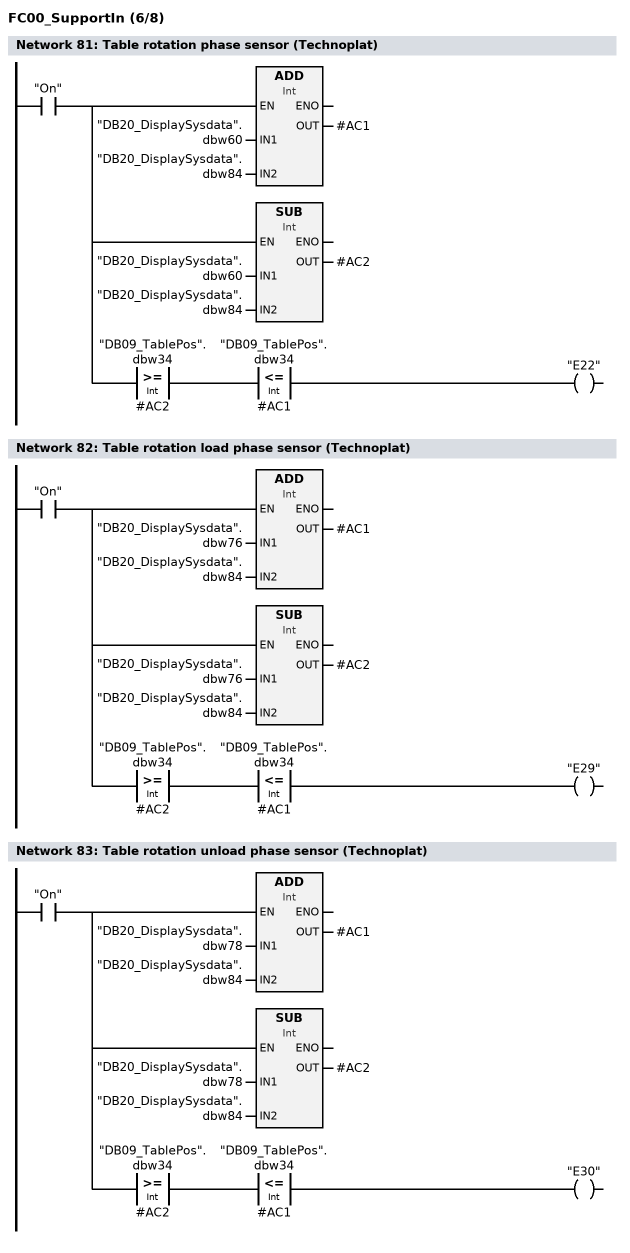
   RUNG wire#powerrail
      Contact( "On" )
      wire#w1
      { S7_Templates := "SrcType := Int"; S7_GenerateENO := "TRUE" } Add(in1 := "DB20_DisplaySysdata".dbw60, in2 := "DB20_DisplaySysdata".dbw84, out => #AC1)
   END_RUNG
   RUNG wire#w1
      { S7_Templates := "SrcType := Int"; S7_GenerateENO := "TRUE" } Sub(in1 := "DB20_DisplaySysdata".dbw60, in2 := "DB20_DisplaySysdata".dbw84, out => #AC2)
   END_RUNG
   RUNG wire#w1
      { S7_Templates := "SrcType := Int" } GE_Contact(in1 := "DB09_TablePos".dbw34, in2 := #AC2)
      { S7_Templates := "SrcType := Int" } LE_Contact(in1 := "DB09_TablePos".dbw34, in2 := #AC1)
      Coil( "E22" )
   END_RUNG
   // the same network as SCL:
   IF "On" THEN
       #AC1 := "DB20_DisplaySysdata".dbw60 + "DB20_DisplaySysdata".dbw84;
       #AC2 := "DB20_DisplaySysdata".dbw60 - "DB20_DisplaySysdata".dbw84;
   END_IF;
   "E22" := "On" AND ("DB09_TablePos".dbw34 >= #AC2) AND ("DB09_TablePos".dbw34 <= #AC1);
END_REGION

REGION Network 82: Table rotation load phase sensor (Technoplat)
   RUNG wire#powerrail
      Contact( "On" )
      wire#w1
      { S7_Templates := "SrcType := Int"; S7_GenerateENO := "TRUE" } Add(in1 := "DB20_DisplaySysdata".dbw76, in2 := "DB20_DisplaySysdata".dbw84, out => #AC1)
   END_RUNG
   RUNG wire#w1
      { S7_Templates := "SrcType := Int"; S7_GenerateENO := "TRUE" } Sub(in1 := "DB20_DisplaySysdata".dbw76, in2 := "DB20_DisplaySysdata".dbw84, out => #AC2)
   END_RUNG
   RUNG wire#w1
      { S7_Templates := "SrcType := Int" } GE_Contact(in1 := "DB09_TablePos".dbw34, in2 := #AC2)
      { S7_Templates := "SrcType := Int" } LE_Contact(in1 := "DB09_TablePos".dbw34, in2 := #AC1)
      Coil( "E29" )
   END_RUNG
   // the same network as SCL:
   IF "On" THEN
       #AC1 := "DB20_DisplaySysdata".dbw76 + "DB20_DisplaySysdata".dbw84;
       #AC2 := "DB20_DisplaySysdata".dbw76 - "DB20_DisplaySysdata".dbw84;
   END_IF;
   "E29" := "On" AND ("DB09_TablePos".dbw34 >= #AC2) AND ("DB09_TablePos".dbw34 <= #AC1);
END_REGION

REGION Network 83: Table rotation unload phase sensor (Technoplat)
   RUNG wire#powerrail
      Contact( "On" )
      wire#w1
      { S7_Templates := "SrcType := Int"; S7_GenerateENO := "TRUE" } Add(in1 := "DB20_DisplaySysdata".dbw78, in2 := "DB20_DisplaySysdata".dbw84, out => #AC1)
   END_RUNG
   RUNG wire#w1
      { S7_Templates := "SrcType := Int"; S7_GenerateENO := "TRUE" } Sub(in1 := "DB20_DisplaySysdata".dbw78, in2 := "DB20_DisplaySysdata".dbw84, out => #AC2)
   END_RUNG
   RUNG wire#w1
      { S7_Templates := "SrcType := Int" } GE_Contact(in1 := "DB09_TablePos".dbw34, in2 := #AC2)
      { S7_Templates := "SrcType := Int" } LE_Contact(in1 := "DB09_TablePos".dbw34, in2 := #AC1)
      Coil( "E30" )
   END_RUNG
   // the same network as SCL:
   IF "On" THEN
       #AC1 := "DB20_DisplaySysdata".dbw78 + "DB20_DisplaySysdata".dbw84;
       #AC2 := "DB20_DisplaySysdata".dbw78 - "DB20_DisplaySysdata".dbw84;
   END_IF;
   "E30" := "On" AND ("DB09_TablePos".dbw34 >= #AC2) AND ("DB09_TablePos".dbw34 <= #AC1);
END_REGION

REGION Network 84: Table rotation phase sensor (Technoplat)
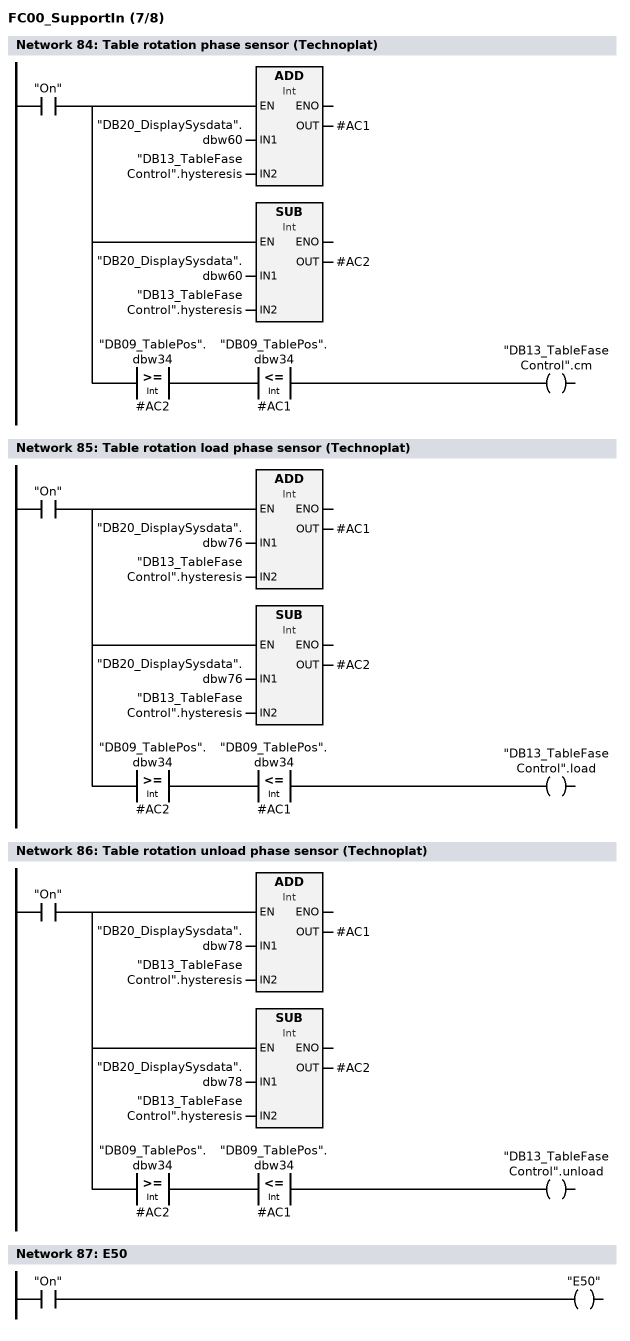
   RUNG wire#powerrail
      Contact( "On" )
      wire#w1
      { S7_Templates := "SrcType := Int"; S7_GenerateENO := "TRUE" } Add(in1 := "DB20_DisplaySysdata".dbw60, in2 := "DB13_TableFaseControl".hysteresis, out => #AC1)
   END_RUNG
   RUNG wire#w1
      { S7_Templates := "SrcType := Int"; S7_GenerateENO := "TRUE" } Sub(in1 := "DB20_DisplaySysdata".dbw60, in2 := "DB13_TableFaseControl".hysteresis, out => #AC2)
   END_RUNG
   RUNG wire#w1
      { S7_Templates := "SrcType := Int" } GE_Contact(in1 := "DB09_TablePos".dbw34, in2 := #AC2)
      { S7_Templates := "SrcType := Int" } LE_Contact(in1 := "DB09_TablePos".dbw34, in2 := #AC1)
      Coil( "DB13_TableFaseControl".cm )
   END_RUNG
   // the same network as SCL:
   IF "On" THEN
       #AC1 := "DB20_DisplaySysdata".dbw60 + "DB13_TableFaseControl".hysteresis;
       #AC2 := "DB20_DisplaySysdata".dbw60 - "DB13_TableFaseControl".hysteresis;
   END_IF;
   "DB13_TableFaseControl".cm := "On" AND ("DB09_TablePos".dbw34 >= #AC2) AND ("DB09_TablePos".dbw34 <= #AC1);
END_REGION

REGION Network 85: Table rotation load phase sensor (Technoplat)
   RUNG wire#powerrail
      Contact( "On" )
      wire#w1
      { S7_Templates := "SrcType := Int"; S7_GenerateENO := "TRUE" } Add(in1 := "DB20_DisplaySysdata".dbw76, in2 := "DB13_TableFaseControl".hysteresis, out => #AC1)
   END_RUNG
   RUNG wire#w1
      { S7_Templates := "SrcType := Int"; S7_GenerateENO := "TRUE" } Sub(in1 := "DB20_DisplaySysdata".dbw76, in2 := "DB13_TableFaseControl".hysteresis, out => #AC2)
   END_RUNG
   RUNG wire#w1
      { S7_Templates := "SrcType := Int" } GE_Contact(in1 := "DB09_TablePos".dbw34, in2 := #AC2)
      { S7_Templates := "SrcType := Int" } LE_Contact(in1 := "DB09_TablePos".dbw34, in2 := #AC1)
      Coil( "DB13_TableFaseControl".load )
   END_RUNG
   // the same network as SCL:
   IF "On" THEN
       #AC1 := "DB20_DisplaySysdata".dbw76 + "DB13_TableFaseControl".hysteresis;
       #AC2 := "DB20_DisplaySysdata".dbw76 - "DB13_TableFaseControl".hysteresis;
   END_IF;
   "DB13_TableFaseControl".load := "On" AND ("DB09_TablePos".dbw34 >= #AC2) AND ("DB09_TablePos".dbw34 <= #AC1);
END_REGION

REGION Network 86: Table rotation unload phase sensor (Technoplat)
   RUNG wire#powerrail
      Contact( "On" )
      wire#w1
      { S7_Templates := "SrcType := Int"; S7_GenerateENO := "TRUE" } Add(in1 := "DB20_DisplaySysdata".dbw78, in2 := "DB13_TableFaseControl".hysteresis, out => #AC1)
   END_RUNG
   RUNG wire#w1
      { S7_Templates := "SrcType := Int"; S7_GenerateENO := "TRUE" } Sub(in1 := "DB20_DisplaySysdata".dbw78, in2 := "DB13_TableFaseControl".hysteresis, out => #AC2)
   END_RUNG
   RUNG wire#w1
      { S7_Templates := "SrcType := Int" } GE_Contact(in1 := "DB09_TablePos".dbw34, in2 := #AC2)
      { S7_Templates := "SrcType := Int" } LE_Contact(in1 := "DB09_TablePos".dbw34, in2 := #AC1)
      Coil( "DB13_TableFaseControl".unload )
   END_RUNG
   // the same network as SCL:
   IF "On" THEN
       #AC1 := "DB20_DisplaySysdata".dbw78 + "DB13_TableFaseControl".hysteresis;
       #AC2 := "DB20_DisplaySysdata".dbw78 - "DB13_TableFaseControl".hysteresis;
   END_IF;
   "DB13_TableFaseControl".unload := "On" AND ("DB09_TablePos".dbw34 >= #AC2) AND ("DB09_TablePos".dbw34 <= #AC1);
END_REGION

REGION Network 87: E50
   RUNG wire#powerrail
      Contact( "On" )
      Coil( "E50" )
   END_RUNG
   // the same network as SCL:
   "E50" := "On";
END_REGION

REGION Network 88: OLD (NOT USED)
END_REGION

REGION Network 89: Key selector automatic (0)/manual (1) mode (Technoplat)
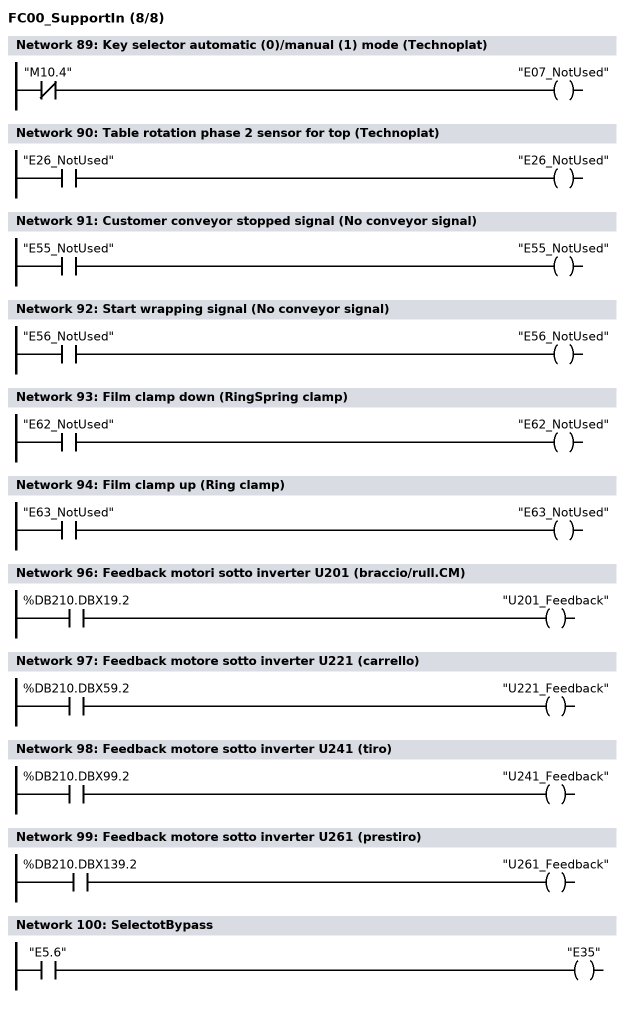
   RUNG wire#powerrail
      I_Contact( "M10.4" )
      Coil( "E07_NotUsed" )
   END_RUNG
   // the same network as SCL:
   "E07_NotUsed" := NOT "M10.4";
END_REGION

REGION Network 90: Table rotation phase 2 sensor for top (Technoplat)
   RUNG wire#powerrail
      Contact( "E26_NotUsed" )
      Coil( "E26_NotUsed" )
   END_RUNG
   // the same network as SCL:
   "E26_NotUsed" := "E26_NotUsed";
END_REGION

REGION Network 91: Customer conveyor stopped signal (No conveyor signal)
   RUNG wire#powerrail
      Contact( "E55_NotUsed" )
      Coil( "E55_NotUsed" )
   END_RUNG
   // the same network as SCL:
   "E55_NotUsed" := "E55_NotUsed";
END_REGION

REGION Network 92: Start wrapping signal (No conveyor signal)
   RUNG wire#powerrail
      Contact( "E56_NotUsed" )
      Coil( "E56_NotUsed" )
   END_RUNG
   // the same network as SCL:
   "E56_NotUsed" := "E56_NotUsed";
END_REGION

REGION Network 93: Film clamp down (RingSpring clamp)
   RUNG wire#powerrail
      Contact( "E62_NotUsed" )
      Coil( "E62_NotUsed" )
   END_RUNG
   // the same network as SCL:
   "E62_NotUsed" := "E62_NotUsed";
END_REGION

REGION Network 94: Film clamp up (Ring clamp)
   RUNG wire#powerrail
      Contact( "E63_NotUsed" )
      Coil( "E63_NotUsed" )
   END_RUNG
   // the same network as SCL:
   "E63_NotUsed" := "E63_NotUsed";
END_REGION

REGION Network 95: PROFINET DATA (inverter)
END_REGION

REGION Network 96: Feedback motori sotto inverter U201 (braccio/rull.CM)
   RUNG wire#powerrail
      Contact( %DB210.DBX19.2 )
      Coil( "U201_Feedback" )
   END_RUNG
   // the same network as SCL:
   "U201_Feedback" := %DB210.DBX19.2;
END_REGION

REGION Network 97: Feedback motore sotto inverter U221 (carrello)
   RUNG wire#powerrail
      Contact( %DB210.DBX59.2 )
      Coil( "U221_Feedback" )
   END_RUNG
   // the same network as SCL:
   "U221_Feedback" := %DB210.DBX59.2;
END_REGION

REGION Network 98: Feedback motore sotto inverter U241 (tiro)
   RUNG wire#powerrail
      Contact( %DB210.DBX99.2 )
      Coil( "U241_Feedback" )
   END_RUNG
   // the same network as SCL:
   "U241_Feedback" := %DB210.DBX99.2;
END_REGION

REGION Network 99: Feedback motore sotto inverter U261 (prestiro)
   RUNG wire#powerrail
      Contact( %DB210.DBX139.2 )
      Coil( "U261_Feedback" )
   END_RUNG
   // the same network as SCL:
   "U261_Feedback" := %DB210.DBX139.2;
END_REGION

REGION Network 100: SelectotBypass
   RUNG wire#powerrail
      Contact( "E5.6" )
      Coil( "E35" )
   END_RUNG
   // the same network as SCL:
   "E35" := "E5.6";
END_REGION
END_FUNCTION

FUNCTION "FC04_TechnoplatAlarm" : Void   // FC4, LAD
TITLE = Alarm for the machine
{ S7_Optimized_Access := 'FALSE' }
AUTHOR : Robopac
VERSION : 0.0
// stored: AutoNumber false, IsIECCheckEnabled false, SetENOAutomatically false, UDAEnableTagReadback false
BEGIN

REGION Network 1: Alarm 1: Pressure switch (Technoplat)
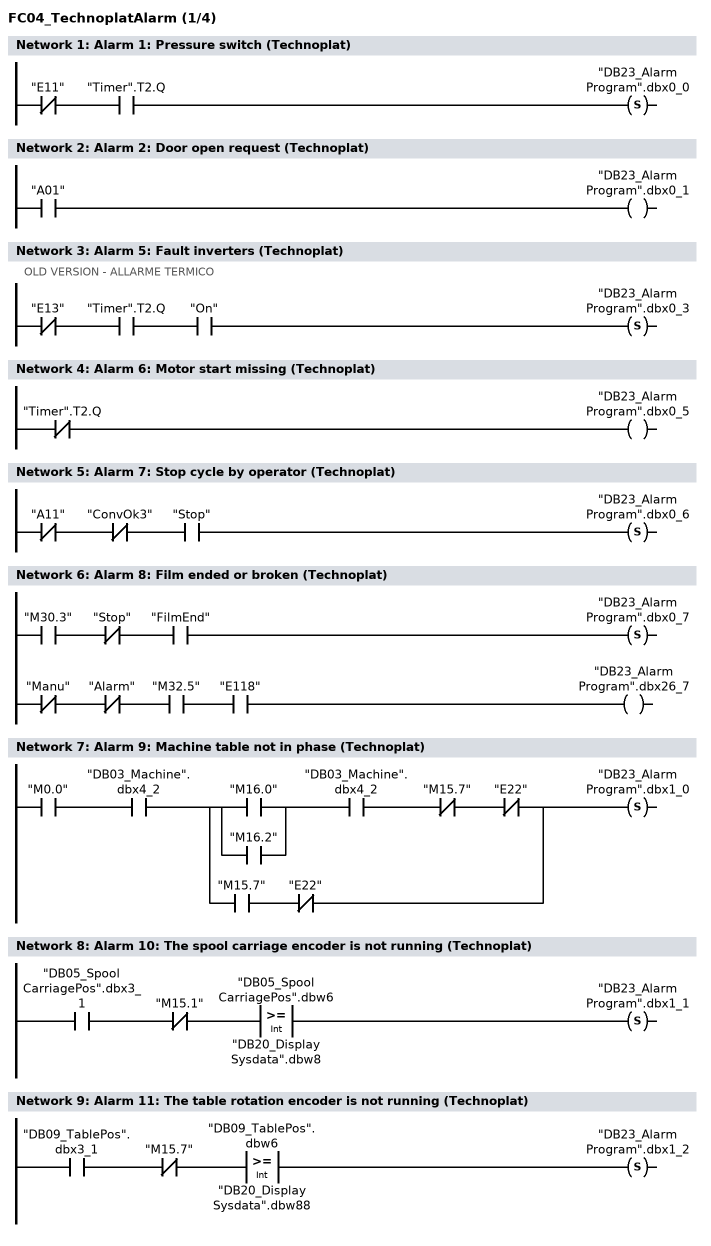
   RUNG wire#powerrail
      I_Contact( "E11" )
      Contact( "Timer".T2.Q )
      S_Coil( "DB23_AlarmProgram".dbx0_0 )
   END_RUNG
   // the same network as SCL:
   IF NOT "E11" AND "Timer".T2.Q THEN "DB23_AlarmProgram".dbx0_0 := TRUE; END_IF;
END_REGION

REGION Network 2: Alarm 2: Door open request (Technoplat)
   RUNG wire#powerrail
      Contact( "A01" )
      Coil( "DB23_AlarmProgram".dbx0_1 )
   END_RUNG
   // the same network as SCL:
   "DB23_AlarmProgram".dbx0_1 := "A01";
END_REGION

REGION Network 3: Alarm 5: Fault inverters (Technoplat)
   // OLD VERSION - ALLARME TERMICO
   RUNG wire#powerrail
      I_Contact( "E13" )
      Contact( "Timer".T2.Q )
      Contact( "On" )
      S_Coil( "DB23_AlarmProgram".dbx0_3 )
   END_RUNG
   // the same network as SCL:
   IF NOT "E13" AND "Timer".T2.Q AND "On" THEN "DB23_AlarmProgram".dbx0_3 := TRUE; END_IF;
END_REGION

REGION Network 4: Alarm 6: Motor start missing (Technoplat)
   RUNG wire#powerrail
      I_Contact( "Timer".T2.Q )
      Coil( "DB23_AlarmProgram".dbx0_5 )
   END_RUNG
   // the same network as SCL:
   "DB23_AlarmProgram".dbx0_5 := NOT "Timer".T2.Q;
END_REGION

REGION Network 5: Alarm 7: Stop cycle by operator (Technoplat)
   RUNG wire#powerrail
      I_Contact( "A11" )
      I_Contact( "ConvOk3" )
      Contact( "Stop" )
      S_Coil( "DB23_AlarmProgram".dbx0_6 )
   END_RUNG
   // the same network as SCL:
   IF NOT "A11" AND NOT "ConvOk3" AND "Stop" THEN "DB23_AlarmProgram".dbx0_6 := TRUE; END_IF;
END_REGION

REGION Network 6: Alarm 8: Film ended or broken (Technoplat)
   RUNG wire#powerrail
      Contact( "M30.3" )
      I_Contact( "Stop" )
      Contact( "FilmEnd" )
      S_Coil( "DB23_AlarmProgram".dbx0_7 )
   END_RUNG
   RUNG wire#powerrail
      I_Contact( "Manu" )
      I_Contact( "Alarm" )
      Contact( "M32.5" )
      Contact( "E118" )
      Coil( "DB23_AlarmProgram".dbx26_7 )
   END_RUNG
   // the same network as SCL:
   IF "M30.3" AND NOT "Stop" AND "FilmEnd" THEN "DB23_AlarmProgram".dbx0_7 := TRUE; END_IF;
   "DB23_AlarmProgram".dbx26_7 := NOT "Manu" AND NOT "Alarm" AND "M32.5" AND "E118";
END_REGION

REGION Network 7: Alarm 9: Machine table not in phase (Technoplat)
   RUNG wire#powerrail
      Contact( "M0.0" )
      Contact( "DB03_Machine".dbx4_2 )
      wire#w1
      Contact( "M16.0" )
      wire#w2
      Contact( "DB03_Machine".dbx4_2 )
      I_Contact( "M15.7" )
      I_Contact( "E22" )
      wire#w3
      S_Coil( "DB23_AlarmProgram".dbx1_0 )
   END_RUNG
   RUNG wire#w1
      Contact( "M16.2" )
   END_RUNG wire#w2
   RUNG wire#w1
      Contact( "M15.7" )
      I_Contact( "E22" )
   END_RUNG wire#w3
   // the same network as SCL:
   IF "M0.0" AND "DB03_Machine".dbx4_2 AND ((("M16.0" OR "M16.2") AND "DB03_Machine".dbx4_2 AND NOT "M15.7" AND NOT "E22") OR ("M15.7" AND NOT "E22")) THEN
       "DB23_AlarmProgram".dbx1_0 := TRUE;
   END_IF;
END_REGION

REGION Network 8: Alarm 10: The spool carriage encoder is not running (Technoplat)
   RUNG wire#powerrail
      Contact( "DB05_SpoolCarriagePos".dbx3_1 )
      I_Contact( "M15.1" )
      { S7_Templates := "SrcType := Int" } GE_Contact(in1 := "DB05_SpoolCarriagePos".dbw6, in2 := "DB20_DisplaySysdata".dbw8)
      S_Coil( "DB23_AlarmProgram".dbx1_1 )
   END_RUNG
   // the same network as SCL:
   IF "DB05_SpoolCarriagePos".dbx3_1 AND NOT "M15.1" AND ("DB05_SpoolCarriagePos".dbw6 >= "DB20_DisplaySysdata".dbw8) THEN
       "DB23_AlarmProgram".dbx1_1 := TRUE;
   END_IF;
END_REGION

REGION Network 9: Alarm 11: The table rotation encoder is not running (Technoplat)
   RUNG wire#powerrail
      Contact( "DB09_TablePos".dbx3_1 )
      I_Contact( "M15.7" )
      { S7_Templates := "SrcType := Int" } GE_Contact(in1 := "DB09_TablePos".dbw6, in2 := "DB20_DisplaySysdata".dbw88)
      S_Coil( "DB23_AlarmProgram".dbx1_2 )
   END_RUNG
   // the same network as SCL:
   IF "DB09_TablePos".dbx3_1 AND NOT "M15.7" AND ("DB09_TablePos".dbw6 >= "DB20_DisplaySysdata".dbw88) THEN
       "DB23_AlarmProgram".dbx1_2 := TRUE;
   END_IF;
END_REGION

REGION Network 10: Alarm 12: Overspeed for arm rotation (Technoplat)
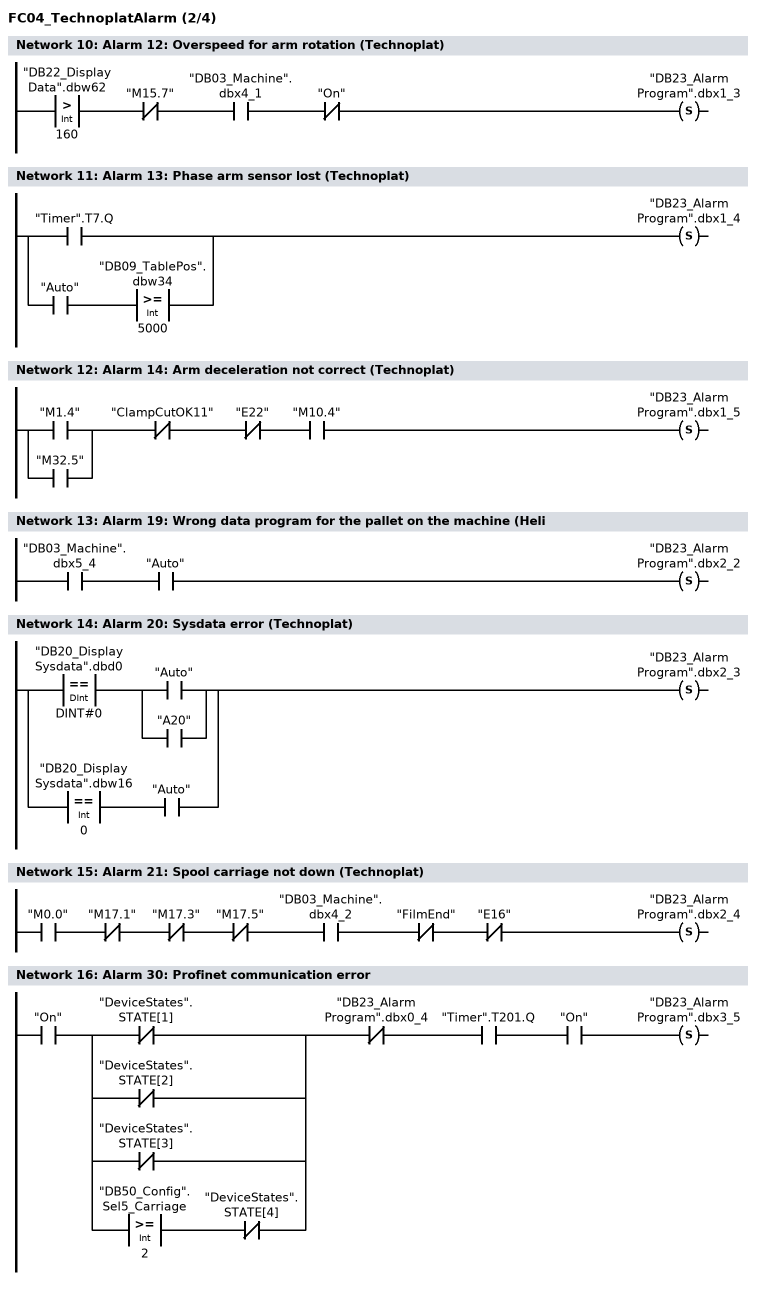
   RUNG wire#powerrail
      { S7_Templates := "SrcType := Int" } GT_Contact(in1 := "DB22_DisplayData".dbw62, in2 := 160)
      I_Contact( "M15.7" )
      Contact( "DB03_Machine".dbx4_1 )
      I_Contact( "On" )
      S_Coil( "DB23_AlarmProgram".dbx1_3 )
   END_RUNG
   // the same network as SCL:
   IF ("DB22_DisplayData".dbw62 > 160) AND NOT "M15.7" AND "DB03_Machine".dbx4_1 AND NOT "On" THEN
       "DB23_AlarmProgram".dbx1_3 := TRUE;
   END_IF;
END_REGION

REGION Network 11: Alarm 13: Phase arm sensor lost (Technoplat)
   RUNG wire#powerrail
      Contact( "Timer".T7.Q )
      wire#w1
      S_Coil( "DB23_AlarmProgram".dbx1_4 )
   END_RUNG
   RUNG wire#powerrail
      Contact( "Auto" )
      { S7_Templates := "SrcType := Int" } GE_Contact(in1 := "DB09_TablePos".dbw34, in2 := 5000)
   END_RUNG wire#w1
   // the same network as SCL:
   IF "Timer".T7.Q OR ("Auto" AND ("DB09_TablePos".dbw34 >= 5000)) THEN
       "DB23_AlarmProgram".dbx1_4 := TRUE;
   END_IF;
END_REGION

REGION Network 12: Alarm 14: Arm deceleration not correct (Technoplat)
   RUNG wire#powerrail
      Contact( "M1.4" )
      wire#w1
      I_Contact( "ClampCutOK11" )
      I_Contact( "E22" )
      Contact( "M10.4" )
      S_Coil( "DB23_AlarmProgram".dbx1_5 )
   END_RUNG
   RUNG wire#powerrail
      Contact( "M32.5" )
   END_RUNG wire#w1
   // the same network as SCL:
   IF ("M1.4" OR "M32.5") AND NOT "ClampCutOK11" AND NOT "E22" AND "M10.4" THEN
       "DB23_AlarmProgram".dbx1_5 := TRUE;
   END_IF;
END_REGION

REGION Network 13: Alarm 19: Wrong data program for the pallet on the machine (Heli
   RUNG wire#powerrail
      Contact( "DB03_Machine".dbx5_4 )
      Contact( "Auto" )
      S_Coil( "DB23_AlarmProgram".dbx2_2 )
   END_RUNG
   // the same network as SCL:
   IF "DB03_Machine".dbx5_4 AND "Auto" THEN "DB23_AlarmProgram".dbx2_2 := TRUE; END_IF;
END_REGION

REGION Network 14: Alarm 20: Sysdata error (Technoplat)
   RUNG wire#powerrail
      { S7_Templates := "SrcType := DInt" } EQ_Contact(in1 := "DB20_DisplaySysdata".dbd0, in2 := DINT#0)
      wire#w1
      Contact( "Auto" )
      wire#w2
      S_Coil( "DB23_AlarmProgram".dbx2_3 )
   END_RUNG
   RUNG wire#w1
      Contact( "A20" )
   END_RUNG wire#w2
   RUNG wire#powerrail
      { S7_Templates := "SrcType := Int" } EQ_Contact(in1 := "DB20_DisplaySysdata".dbw16, in2 := 0)
      Contact( "Auto" )
   END_RUNG wire#w2
   // the same network as SCL:
   IF (("DB20_DisplaySysdata".dbd0 = DINT#0) AND ("Auto" OR "A20")) OR (("DB20_DisplaySysdata".dbw16 = 0) AND "Auto") THEN
       "DB23_AlarmProgram".dbx2_3 := TRUE;
   END_IF;
END_REGION

REGION Network 15: Alarm 21: Spool carriage not down (Technoplat)
   RUNG wire#powerrail
      Contact( "M0.0" )
      I_Contact( "M17.1" )
      I_Contact( "M17.3" )
      I_Contact( "M17.5" )
      Contact( "DB03_Machine".dbx4_2 )
      I_Contact( "FilmEnd" )
      I_Contact( "E16" )
      S_Coil( "DB23_AlarmProgram".dbx2_4 )
   END_RUNG
   // the same network as SCL:
   IF "M0.0" AND NOT "M17.1" AND NOT "M17.3" AND NOT "M17.5" AND "DB03_Machine".dbx4_2 AND NOT "FilmEnd" AND NOT "E16" THEN
       "DB23_AlarmProgram".dbx2_4 := TRUE;
   END_IF;
END_REGION

REGION Network 16: Alarm 30: Profinet communication error
   RUNG wire#powerrail
      Contact( "On" )
      wire#w1
      I_Contact( "DeviceStates".STATE[1] )
      wire#w2
      I_Contact( "DB23_AlarmProgram".dbx0_4 )
      Contact( "Timer".T201.Q )
      Contact( "On" )
      S_Coil( "DB23_AlarmProgram".dbx3_5 )
   END_RUNG
   RUNG wire#w1
      I_Contact( "DeviceStates".STATE[2] )
   END_RUNG wire#w2
   RUNG wire#w1
      I_Contact( "DeviceStates".STATE[3] )
   END_RUNG wire#w2
   RUNG wire#w1
      { S7_Templates := "SrcType := Int" } GE_Contact(in1 := "DB50_Config".Sel5_Carriage, in2 := 2)
      I_Contact( "DeviceStates".STATE[4] )
   END_RUNG wire#w2
   // the same network as SCL:
   IF "On" AND (NOT "DeviceStates".STATE[1] OR NOT "DeviceStates".STATE[2] OR NOT "DeviceStates".STATE[3] OR (("DB50_Config".Sel5_Carriage >= 2) AND NOT "DeviceStates".STATE[4])) AND NOT "DB23_AlarmProgram".dbx0_4 AND "Timer".T201.Q AND "On" THEN
       "DB23_AlarmProgram".dbx3_5 := TRUE;
   END_IF;
END_REGION

REGION Network 17: Alarm 31: Modbus communication error
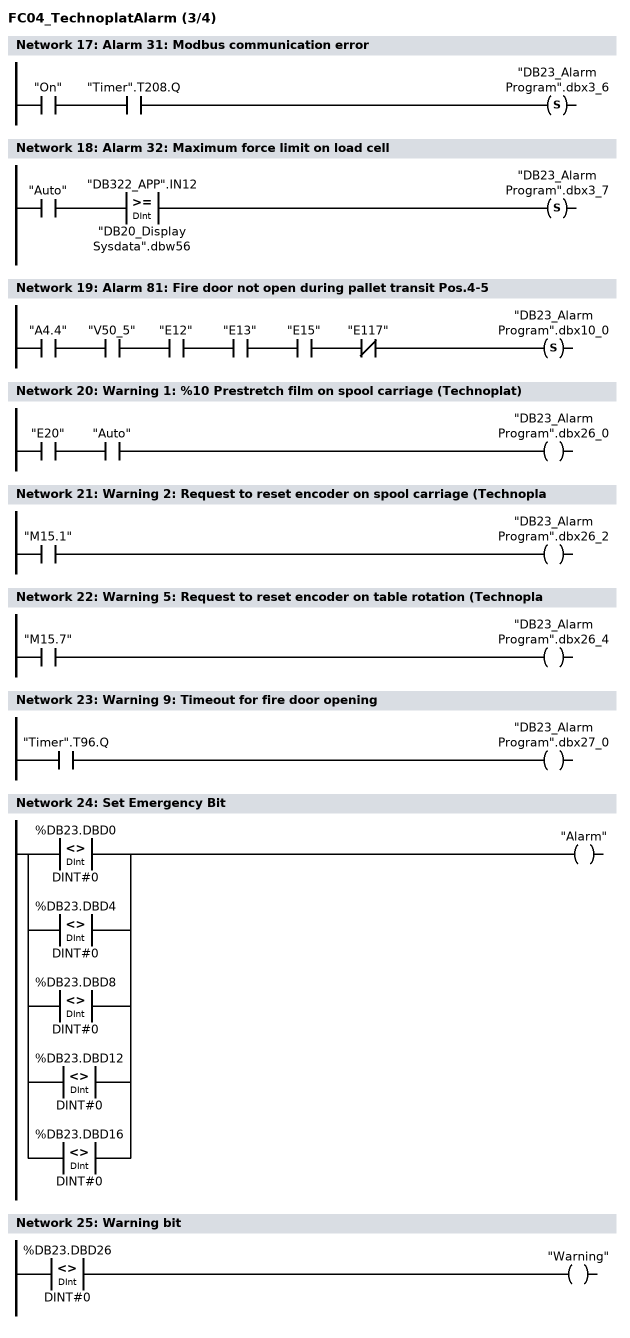
   RUNG wire#powerrail
      Contact( "On" )
      Contact( "Timer".T208.Q )
      S_Coil( "DB23_AlarmProgram".dbx3_6 )
   END_RUNG
   // the same network as SCL:
   IF "On" AND "Timer".T208.Q THEN "DB23_AlarmProgram".dbx3_6 := TRUE; END_IF;
END_REGION

REGION Network 18: Alarm 32: Maximum force limit on load cell
   RUNG wire#powerrail
      Contact( "Auto" )
      { S7_Templates := "SrcType := DInt" } GE_Contact(in1 := "DB322_APP".IN12, in2 := "DB20_DisplaySysdata".dbw56)
      S_Coil( "DB23_AlarmProgram".dbx3_7 )
   END_RUNG
   // the same network as SCL:
   IF "Auto" AND ("DB322_APP".IN12 >= "DB20_DisplaySysdata".dbw56) THEN
       "DB23_AlarmProgram".dbx3_7 := TRUE;
   END_IF;
END_REGION

REGION Network 19: Alarm 81: Fire door not open during pallet transit Pos.4-5
   RUNG wire#powerrail
      Contact( "A4.4" )
      Contact( "V50_5" )
      Contact( "E12" )
      Contact( "E13" )
      Contact( "E15" )
      I_Contact( "E117" )
      S_Coil( "DB23_AlarmProgram".dbx10_0 )
   END_RUNG
   // the same network as SCL:
   IF "A4.4" AND "V50_5" AND "E12" AND "E13" AND "E15" AND NOT "E117" THEN
       "DB23_AlarmProgram".dbx10_0 := TRUE;
   END_IF;
END_REGION

REGION Network 20: Warning 1: %10 Prestretch film on spool carriage (Technoplat)
   RUNG wire#powerrail
      Contact( "E20" )
      Contact( "Auto" )
      Coil( "DB23_AlarmProgram".dbx26_0 )
   END_RUNG
   // the same network as SCL:
   "DB23_AlarmProgram".dbx26_0 := "E20" AND "Auto";
END_REGION

REGION Network 21: Warning 2: Request to reset encoder on spool carriage (Technopla
   RUNG wire#powerrail
      Contact( "M15.1" )
      Coil( "DB23_AlarmProgram".dbx26_2 )
   END_RUNG
   // the same network as SCL:
   "DB23_AlarmProgram".dbx26_2 := "M15.1";
END_REGION

REGION Network 22: Warning 5: Request to reset encoder on table rotation (Technopla
   RUNG wire#powerrail
      Contact( "M15.7" )
      Coil( "DB23_AlarmProgram".dbx26_4 )
   END_RUNG
   // the same network as SCL:
   "DB23_AlarmProgram".dbx26_4 := "M15.7";
END_REGION

REGION Network 23: Warning 9: Timeout for fire door opening
   RUNG wire#powerrail
      Contact( "Timer".T96.Q )
      Coil( "DB23_AlarmProgram".dbx27_0 )
   END_RUNG
   // the same network as SCL:
   "DB23_AlarmProgram".dbx27_0 := "Timer".T96.Q;
END_REGION

REGION Network 24: Set Emergency Bit
   RUNG wire#powerrail
      { S7_Templates := "SrcType := DInt" } NE_Contact(in1 := %DB23.DBD0, in2 := DINT#0)
      wire#w1
      Coil( "Alarm" )
   END_RUNG
   RUNG wire#powerrail
      { S7_Templates := "SrcType := DInt" } NE_Contact(in1 := %DB23.DBD4, in2 := DINT#0)
   END_RUNG wire#w1
   RUNG wire#powerrail
      { S7_Templates := "SrcType := DInt" } NE_Contact(in1 := %DB23.DBD8, in2 := DINT#0)
   END_RUNG wire#w1
   RUNG wire#powerrail
      { S7_Templates := "SrcType := DInt" } NE_Contact(in1 := %DB23.DBD12, in2 := DINT#0)
   END_RUNG wire#w1
   RUNG wire#powerrail
      { S7_Templates := "SrcType := DInt" } NE_Contact(in1 := %DB23.DBD16, in2 := DINT#0)
   END_RUNG wire#w1
   // the same network as SCL:
   "Alarm" := (%DB23.DBD0 <> DINT#0) OR (%DB23.DBD4 <> DINT#0) OR (%DB23.DBD8 <> DINT#0) OR (%DB23.DBD12 <> DINT#0) OR (%DB23.DBD16 <> DINT#0);
END_REGION

REGION Network 25: Warning bit
   RUNG wire#powerrail
      { S7_Templates := "SrcType := DInt" } NE_Contact(in1 := %DB23.DBD26, in2 := DINT#0)
      Coil( "Warning" )
   END_RUNG
   // the same network as SCL:
   "Warning" := %DB23.DBD26 <> DINT#0;
END_REGION

REGION Network 26: First cycle
